(* CODESYS project mobject-graph-math-pack.library
   Company: mobject
   DefaultNamespace: mobject-graph-math-pack
   Version: 0.1.0
   Placeholder: mobject-graph-math-pack
   Author: mobject dev team
   Title: mobject-graph-math-pack

Project tree, tasks and I/O mapping:
  libraries: mobject-core, 0.7.0 (mobject); mobject-graph, 0.16.0 (mobject); Tc2_Math, * (Beckhoff Automation GmbH); Tc2_Standard, * (Beckhoff Automation GmbH); Tc2_System, * (Beckhoff Automation GmbH); Tc2_Utilities, * (Beckhoff Automation GmbH); Tc3_Module, * (Beckhoff Automation GmbH)
  Advanced/
    Nodes/
      ABS/
        function block ABS_BYTE [ST]: FB_init, Clone, OnExecute
        function block ABS_DINT [ST]: FB_init, Clone, OnExecute
        function block ABS_DWORD [ST]: FB_init, Clone, OnExecute
        function block ABS_INT [ST]: FB_init, Clone, OnExecute
        function block ABS_LINT [ST]: FB_init, Clone, OnExecute
        function block ABS_LREAL [ST]: FB_init, Clone, OnExecute
        function block ABS_LWORD [ST]: FB_init, Clone, OnExecute
        function block ABS_REAL [ST]: FB_init, Clone, OnExecute
        function block ABS_SINT [ST]: FB_init, Clone, OnExecute
        function block ABS_UDINT [ST]: FB_init, Clone, OnExecute
        function block ABS_UINT [ST]: FB_init, Clone, OnExecute
        function block ABS_ULINT [ST]: FB_init, Clone, OnExecute
        function block ABS_USINT [ST]: FB_init, Clone, OnExecute
        function block ABS_WORD [ST]: FB_init, Clone, OnExecute
      ACOS/
        function block ACOS_LREAL [ST]: FB_init, Clone, OnExecute
      ASIN/
        function block ASIN_LREAL [ST]: FB_init, Clone, OnExecute
      ATAN/
        function block ATAN_LREAL [ST]: FB_init, Clone, OnExecute
      COS/
        function block COS_LREAL [ST]: FB_init, Clone, OnExecute
      EXP/
        function block EXP_LREAL [ST]: FB_init, Clone, OnExecute
      EXPT/
        function block EXPT_LREAL [ST]: FB_init, Clone, OnExecute
      FLOOR/
        function block FLOOR_LREAL [ST]: FB_init, Clone, OnExecute
      FRAC/
        function block FRAC_LREAL [ST]: FB_init, Clone, OnExecute
      LN/
        function block LN_LREAL [ST]: FB_init, Clone, OnExecute
      LOG/
        function block LOG_LREAL [ST]: FB_init, Clone, OnExecute
      MODABS/
        function block MODABS_LREAL [ST]: FB_init, Clone, OnExecute
      MODTURNS/
        function block MODTURNS_LREAL [ST]: FB_init, Clone, OnExecute
      SIN/
        function block SIN_LREAL [ST]: FB_init, Clone, OnExecute
      SQRT/
        function block SQRT_LREAL [ST]: FB_init, Clone, OnExecute
      TAN/
        function block TAN_LREAL [ST]: FB_init, Clone, OnExecute
      TRUNC/
        function block TRUNC_LREAL [ST]: FB_init, Clone, OnExecute
      function block MathAdvancedPack [ST]: Register
  Comparison/
    Nodes/
      EQ/
        function block EQ_BYTE [ST]: FB_init, Clone, OnExecute
        function block EQ_DINT [ST]: FB_init, Clone, OnExecute
        function block EQ_DWORD [ST]: FB_init, Clone, OnExecute
        function block EQ_INT [ST]: FB_init, Clone, OnExecute
        function block EQ_LINT [ST]: FB_init, Clone, OnExecute
        function block EQ_LREAL [ST]: FB_init, Clone, OnExecute
        function block EQ_LWORD [ST]: FB_init, Clone, OnExecute
        function block EQ_REAL [ST]: FB_init, Clone, OnExecute
        function block EQ_SINT [ST]: FB_init, Clone, OnExecute
        function block EQ_UDINT [ST]: FB_init, Clone, OnExecute
        function block EQ_UINT [ST]: FB_init, Clone, OnExecute
        function block EQ_ULINT [ST]: FB_init, Clone, OnExecute
        function block EQ_USINT [ST]: FB_init, Clone, OnExecute
        function block EQ_WORD [ST]: FB_init, Clone, OnExecute
      GE/
        function block GE_BYTE [ST]: FB_init, Clone, OnExecute
        function block GE_DINT [ST]: FB_init, Clone, OnExecute
        function block GE_DWORD [ST]: FB_init, Clone, OnExecute
        function block GE_INT [ST]: FB_init, Clone, OnExecute
        function block GE_LINT [ST]: FB_init, Clone, OnExecute
        function block GE_LREAL [ST]: FB_init, Clone, OnExecute
        function block GE_LWORD [ST]: FB_init, Clone, OnExecute
        function block GE_REAL [ST]: FB_init, Clone, OnExecute
        function block GE_SINT [ST]: FB_init, Clone, OnExecute
        function block GE_UDINT [ST]: FB_init, Clone, OnExecute
        function block GE_UINT [ST]: FB_init, Clone, OnExecute
        function block GE_ULINT [ST]: FB_init, Clone, OnExecute
        function block GE_USINT [ST]: FB_init, Clone, OnExecute
        function block GE_WORD [ST]: FB_init, Clone, OnExecute
      GT/
        function block GT_BYTE [ST]: FB_init, Clone, OnExecute
        function block GT_DINT [ST]: FB_init, Clone, OnExecute
        function block GT_DWORD [ST]: FB_init, Clone, OnExecute
        function block GT_INT [ST]: FB_init, Clone, OnExecute
        function block GT_LINT [ST]: FB_init, Clone, OnExecute
        function block GT_LREAL [ST]: FB_init, Clone, OnExecute
        function block GT_LWORD [ST]: FB_init, Clone, OnExecute
        function block GT_REAL [ST]: FB_init, Clone, OnExecute
        function block GT_SINT [ST]: FB_init, Clone, OnExecute
        function block GT_UDINT [ST]: FB_init, Clone, OnExecute
        function block GT_UINT [ST]: FB_init, Clone, OnExecute
        function block GT_ULINT [ST]: FB_init, Clone, OnExecute
        function block GT_USINT [ST]: FB_init, Clone, OnExecute
        function block GT_WORD [ST]: FB_init, Clone, OnExecute
      LE/
        function block LE_BYTE [ST]: FB_init, Clone, OnExecute
        function block LE_DINT [ST]: FB_init, Clone, OnExecute
        function block LE_DWORD [ST]: FB_init, Clone, OnExecute
        function block LE_INT [ST]: FB_init, Clone, OnExecute
        function block LE_LINT [ST]: FB_init, Clone, OnExecute
        function block LE_LREAL [ST]: FB_init, Clone, OnExecute
        function block LE_LWORD [ST]: FB_init, Clone, OnExecute
        function block LE_REAL [ST]: FB_init, Clone, OnExecute
        function block LE_SINT [ST]: FB_init, Clone, OnExecute
        function block LE_UDINT [ST]: FB_init, Clone, OnExecute
        function block LE_UINT [ST]: FB_init, Clone, OnExecute
        function block LE_ULINT [ST]: FB_init, Clone, OnExecute
        function block LE_USINT [ST]: FB_init, Clone, OnExecute
        function block LE_WORD [ST]: FB_init, Clone, OnExecute
      LT/
        function block LT_BYTE [ST]: FB_init, Clone, OnExecute
        function block LT_DINT [ST]: FB_init, Clone, OnExecute
        function block LT_DWORD [ST]: FB_init, Clone, OnExecute
        function block LT_INT [ST]: FB_init, Clone, OnExecute
        function block LT_LINT [ST]: FB_init, Clone, OnExecute
        function block LT_LREAL [ST]: FB_init, Clone, OnExecute
        function block LT_LWORD [ST]: FB_init, Clone, OnExecute
        function block LT_REAL [ST]: FB_init, Clone, OnExecute
        function block LT_SINT [ST]: FB_init, Clone, OnExecute
        function block LT_UDINT [ST]: FB_init, Clone, OnExecute
        function block LT_UINT [ST]: FB_init, Clone, OnExecute
        function block LT_ULINT [ST]: FB_init, Clone, OnExecute
        function block LT_USINT [ST]: FB_init, Clone, OnExecute
        function block LT_WORD [ST]: FB_init, Clone, OnExecute
      NE/
        function block NE_BYTE [ST]: FB_init, Clone, OnExecute
        function block NE_DINT [ST]: FB_init, Clone, OnExecute
        function block NE_DWORD [ST]: FB_init, Clone, OnExecute
        function block NE_INT [ST]: FB_init, Clone, OnExecute
        function block NE_LINT [ST]: FB_init, Clone, OnExecute
        function block NE_LREAL [ST]: FB_init, Clone, OnExecute
        function block NE_LWORD [ST]: FB_init, Clone, OnExecute
        function block NE_REAL [ST]: FB_init, Clone, OnExecute
        function block NE_SINT [ST]: FB_init, Clone, OnExecute
        function block NE_UDINT [ST]: FB_init, Clone, OnExecute
        function block NE_UINT [ST]: FB_init, Clone, OnExecute
        function block NE_ULINT [ST]: FB_init, Clone, OnExecute
        function block NE_USINT [ST]: FB_init, Clone, OnExecute
        function block NE_WORD [ST]: FB_init, Clone, OnExecute
    function block MathComparisonPack [ST]: Register
  Core/
    Nodes/
      ADD/
        function block ADD_BYTE [ST]: FB_init, Clone, OnExecute
        function block ADD_DINT [ST]: FB_init, Clone, OnExecute
        function block ADD_DWORD [ST]: FB_init, Clone, OnExecute
        function block ADD_INT [ST]: FB_init, Clone, OnExecute
        function block ADD_LINT [ST]: FB_init, Clone, OnExecute
        function block ADD_LREAL [ST]: FB_init, Clone, OnExecute
        function block ADD_LWORD [ST]: FB_init, Clone, OnExecute
        function block ADD_REAL [ST]: FB_init, Clone, OnExecute
        function block ADD_SINT [ST]: FB_init, Clone, OnExecute
        function block ADD_UDINT [ST]: FB_init, Clone, OnExecute
        function block ADD_UINT [ST]: FB_init, Clone, OnExecute
        function block ADD_ULINT [ST]: FB_init, Clone, OnExecute
        function block ADD_USINT [ST]: FB_init, Clone, OnExecute
        function block ADD_WORD [ST]: FB_init, Clone, OnExecute
      DIV/
        function block DIV_BYTE [ST]: FB_init, Clone, OnExecute
        function block DIV_DINT [ST]: FB_init, Clone, OnExecute
        function block DIV_DWORD [ST]: FB_init, Clone, OnExecute
        function block DIV_INT [ST]: FB_init, Clone, OnExecute
        function block DIV_LINT [ST]: FB_init, Clone, OnExecute
        function block DIV_LREAL [ST]: FB_init, Clone, OnExecute
        function block DIV_LWORD [ST]: FB_init, Clone, OnExecute
        function block DIV_REAL [ST]: FB_init, Clone, OnExecute
        function block DIV_SINT [ST]: FB_init, Clone, OnExecute
        function block DIV_UDINT [ST]: FB_init, Clone, OnExecute
        function block DIV_UINT [ST]: FB_init, Clone, OnExecute
        function block DIV_ULINT [ST]: FB_init, Clone, OnExecute
        function block DIV_USINT [ST]: FB_init, Clone, OnExecute
        function block DIV_WORD [ST]: FB_init, Clone, OnExecute
      MOD/
        function block MOD_BYTE [ST]: FB_init, Clone, OnExecute
        function block MOD_DINT [ST]: FB_init, Clone, OnExecute
        function block MOD_DWORD [ST]: FB_init, Clone, OnExecute
        function block MOD_INT [ST]: FB_init, Clone, OnExecute
        function block MOD_LINT [ST]: FB_init, Clone, OnExecute
        function block MOD_LREAL [ST]: FB_init, Clone, OnExecute
        function block MOD_LWORD [ST]: FB_init, Clone, OnExecute
        function block MOD_SINT [ST]: FB_init, Clone, OnExecute
        function block MOD_UDINT [ST]: FB_init, Clone, OnExecute
        function block MOD_UINT [ST]: FB_init, Clone, OnExecute
        function block MOD_ULINT [ST]: FB_init, Clone, OnExecute
        function block MOD_USINT [ST]: FB_init, Clone, OnExecute
        function block MOD_WORD [ST]: FB_init, Clone, OnExecute
      MUL/
        function block MUL_BYTE [ST]: FB_init, Clone, OnExecute
        function block MUL_DINT [ST]: FB_init, Clone, OnExecute
        function block MUL_DWORD [ST]: FB_init, Clone, OnExecute
        function block MUL_INT [ST]: FB_init, Clone, OnExecute
        function block MUL_LINT [ST]: FB_init, Clone, OnExecute
        function block MUL_LREAL [ST]: FB_init, Clone, OnExecute
        function block MUL_LWORD [ST]: FB_init, Clone, OnExecute
        function block MUL_REAL [ST]: FB_init, Clone, OnExecute
        function block MUL_SINT [ST]: FB_init, Clone, OnExecute
        function block MUL_UDINT [ST]: FB_init, Clone, OnExecute
        function block MUL_UINT [ST]: FB_init, Clone, OnExecute
        function block MUL_ULINT [ST]: FB_init, Clone, OnExecute
        function block MUL_USINT [ST]: FB_init, Clone, OnExecute
        function block MUL_WORD [ST]: FB_init, Clone, OnExecute
      SUB/
        function block SUB_BYTE [ST]: FB_init, Clone, OnExecute
        function block SUB_DINT [ST]: FB_init, Clone, OnExecute
        function block SUB_DWORD [ST]: FB_init, Clone, OnExecute
        function block SUB_INT [ST]: FB_init, Clone, OnExecute
        function block SUB_LINT [ST]: FB_init, Clone, OnExecute
        function block SUB_LREAL [ST]: FB_init, Clone, OnExecute
        function block SUB_LWORD [ST]: FB_init, Clone, OnExecute
        function block SUB_REAL [ST]: FB_init, Clone, OnExecute
        function block SUB_SINT [ST]: FB_init, Clone, OnExecute
        function block SUB_UDINT [ST]: FB_init, Clone, OnExecute
        function block SUB_UINT [ST]: FB_init, Clone, OnExecute
        function block SUB_ULINT [ST]: FB_init, Clone, OnExecute
        function block SUB_USINT [ST]: FB_init, Clone, OnExecute
        function block SUB_WORD [ST]: FB_init, Clone, OnExecute
    function block MathCorePack [ST]: Register
  Logic/
    Nodes/
      AND/
        function block AND_BOOL [ST]: FB_init, Clone, OnExecute
        function block AND_BYTE [ST]: FB_init, Clone, OnExecute
        function block AND_DINT [ST]: FB_init, Clone, OnExecute
        function block AND_DWORD [ST]: FB_init, Clone, OnExecute
        function block AND_INT [ST]: FB_init, Clone, OnExecute
        function block AND_LINT [ST]: FB_init, Clone, OnExecute
        function block AND_LWORD [ST]: FB_init, Clone, OnExecute
        function block AND_SINT [ST]: FB_init, Clone, OnExecute
        function block AND_UDINT [ST]: FB_init, Clone, OnExecute
        function block AND_UINT [ST]: FB_init, Clone, OnExecute
        function block AND_ULINT [ST]: FB_init, Clone, OnExecute
        function block AND_USINT [ST]: FB_init, Clone, OnExecute
        function block AND_WORD [ST]: FB_init, Clone, OnExecute
      NOT/
        function block NOT_BOOL [ST]: FB_init, Clone, OnExecute
        function block NOT_BYTE [ST]: FB_init, Clone, OnExecute
        function block NOT_DINT [ST]: FB_init, Clone, OnExecute
        function block NOT_DWORD [ST]: FB_init, Clone, OnExecute
        function block NOT_INT [ST]: FB_init, Clone, OnExecute
        function block NOT_LINT [ST]: FB_init, Clone, OnExecute
        function block NOT_LWORD [ST]: FB_init, Clone, OnExecute
        function block NOT_SINT [ST]: FB_init, Clone, OnExecute
        function block NOT_UDINT [ST]: FB_init, Clone, OnExecute
        function block NOT_UINT [ST]: FB_init, Clone, OnExecute
        function block NOT_ULINT [ST]: FB_init, Clone, OnExecute
        function block NOT_USINT [ST]: FB_init, Clone, OnExecute
        function block NOT_WORD [ST]: FB_init, Clone, OnExecute
      OR/
        function block OR_BOOL [ST]: FB_init, Clone, OnExecute
        function block OR_BYTE [ST]: FB_init, Clone, OnExecute
        function block OR_DINT [ST]: FB_init, Clone, OnExecute
        function block OR_DWORD [ST]: FB_init, Clone, OnExecute
        function block OR_INT [ST]: FB_init, Clone, OnExecute
        function block OR_LINT [ST]: FB_init, Clone, OnExecute
        function block OR_LWORD [ST]: FB_init, Clone, OnExecute
        function block OR_SINT [ST]: FB_init, Clone, OnExecute
        function block OR_UDINT [ST]: FB_init, Clone, OnExecute
        function block OR_UINT [ST]: FB_init, Clone, OnExecute
        function block OR_ULINT [ST]: FB_init, Clone, OnExecute
        function block OR_USINT [ST]: FB_init, Clone, OnExecute
        function block OR_WORD [ST]: FB_init, Clone, OnExecute
      XOR/
        function block XOR_BOOL [ST]: FB_init, Clone, OnExecute
        function block XOR_BYTE [ST]: FB_init, Clone, OnExecute
        function block XOR_DINT [ST]: FB_init, Clone, OnExecute
        function block XOR_DWORD [ST]: FB_init, Clone, OnExecute
        function block XOR_INT [ST]: FB_init, Clone, OnExecute
        function block XOR_LINT [ST]: FB_init, Clone, OnExecute
        function block XOR_LWORD [ST]: FB_init, Clone, OnExecute
        function block XOR_SINT [ST]: FB_init, Clone, OnExecute
        function block XOR_UDINT [ST]: FB_init, Clone, OnExecute
        function block XOR_UINT [ST]: FB_init, Clone, OnExecute
        function block XOR_ULINT [ST]: FB_init, Clone, OnExecute
        function block XOR_USINT [ST]: FB_init, Clone, OnExecute
        function block XOR_WORD [ST]: FB_init, Clone, OnExecute
    function block MathLogicPack [ST]: Register
  Selection/
    Nodes/
      MAX/
        function block MAX_BYTE [ST]: FB_init, Clone, OnExecute
        function block MAX_DINT [ST]: FB_init, Clone, OnExecute
        function block MAX_DWORD [ST]: FB_init, Clone, OnExecute
        function block MAX_INT [ST]: FB_init, Clone, OnExecute
        function block MAX_LINT [ST]: FB_init, Clone, OnExecute
        function block MAX_LREAL [ST]: FB_init, Clone, OnExecute
        function block MAX_LWORD [ST]: FB_init, Clone, OnExecute
        function block MAX_REAL [ST]: FB_init, Clone, OnExecute
        function block MAX_SINT [ST]: FB_init, Clone, OnExecute
        function block MAX_UDINT [ST]: FB_init, Clone, OnExecute
        function block MAX_UINT [ST]: FB_init, Clone, OnExecute
        function block MAX_ULINT [ST]: FB_init, Clone, OnExecute
        function block MAX_USINT [ST]: FB_init, Clone, OnExecute
        function block MAX_WORD [ST]: FB_init, Clone, OnExecute
      MIN/
        function block MIN_BYTE [ST]: FB_init, Clone, OnExecute
        function block MIN_DINT [ST]: FB_init, Clone, OnExecute
        function block MIN_DWORD [ST]: FB_init, Clone, OnExecute
        function block MIN_INT [ST]: FB_init, Clone, OnExecute
        function block MIN_LINT [ST]: FB_init, Clone, OnExecute
        function block MIN_LREAL [ST]: FB_init, Clone, OnExecute
        function block MIN_LWORD [ST]: FB_init, Clone, OnExecute
        function block MIN_REAL [ST]: FB_init, Clone, OnExecute
        function block MIN_SINT [ST]: FB_init, Clone, OnExecute
        function block MIN_UDINT [ST]: FB_init, Clone, OnExecute
        function block MIN_UINT [ST]: FB_init, Clone, OnExecute
        function block MIN_ULINT [ST]: FB_init, Clone, OnExecute
        function block MIN_USINT [ST]: FB_init, Clone, OnExecute
        function block MIN_WORD [ST]: FB_init, Clone, OnExecute
      SEL/
        function block SEL_BYTE [ST]: FB_init, Clone, OnExecute
        function block SEL_DINT [ST]: FB_init, Clone, OnExecute
        function block SEL_DWORD [ST]: FB_init, Clone, OnExecute
        function block SEL_INT [ST]: FB_init, Clone, OnExecute
        function block SEL_LINT [ST]: FB_init, Clone, OnExecute
        function block SEL_LREAL [ST]: FB_init, Clone, OnExecute
        function block SEL_LWORD [ST]: FB_init, Clone, OnExecute
        function block SEL_REAL [ST]: FB_init, Clone, OnExecute
        function block SEL_SINT [ST]: FB_init, Clone, OnExecute
        function block SEL_UDINT [ST]: FB_init, Clone, OnExecute
        function block SEL_UINT [ST]: FB_init, Clone, OnExecute
        function block SEL_ULINT [ST]: FB_init, Clone, OnExecute
        function block SEL_USINT [ST]: FB_init, Clone, OnExecute
        function block SEL_WORD [ST]: FB_init, Clone, OnExecute
    function block MathSelectionPack [ST]: Register
  function block MathPack [ST]: Register
*)

// Advanced/Nodes/ABS/ABS_BYTE
{attribute 'linkalways'} 
{attribute 'no_explicit_call' := 'This FB is a CLASS and must be accessed using methods or properties'}
{attribute 'enable_dynamic_creation'}
FUNCTION_BLOCK FINAL ABS_BYTE EXTENDS Node
VAR
	in : _BYTE(0);
	out : _BYTE(0);
END_VAR

METHOD FB_init : BOOL
VAR_INPUT
	bInitRetains : BOOL; // if TRUE, the retain variables are initialized (warm start / cold start)
	bInCopyCode : BOOL;  // if TRUE, the instance afterwards gets moved into the copy code (online change)
END_VAR
AddInput('in',THIS^.in);
AddOutput('out', THIS^.out);
END_METHOD

METHOD PUBLIC Clone : I_Node
VAR
	pNode : POINTER TO ABS_BYTE;
END_VAR
pNode := __NEW(ABS_BYTE);
Clone := pNode^;
END_METHOD

METHOD PROTECTED OnExecute
VAR
END_VAR
out.Value := ABS(in.Value);
END_METHOD

END_FUNCTION_BLOCK

// Advanced/Nodes/ABS/ABS_DINT
{attribute 'linkalways'} 
{attribute 'no_explicit_call' := 'This FB is a CLASS and must be accessed using methods or properties'}
{attribute 'enable_dynamic_creation'}
FUNCTION_BLOCK FINAL ABS_DINT EXTENDS Node
VAR
	in : _DINT(0);
	out : _DINT(0);
END_VAR

METHOD FB_init : BOOL
VAR_INPUT
	bInitRetains : BOOL; // if TRUE, the retain variables are initialized (warm start / cold start)
	bInCopyCode : BOOL;  // if TRUE, the instance afterwards gets moved into the copy code (online change)
END_VAR
AddInput('in',THIS^.in);
AddOutput('out', THIS^.out);
END_METHOD

METHOD PUBLIC Clone : I_Node
VAR
	pNode : POINTER TO ABS_DINT;
END_VAR
pNode := __NEW(ABS_DINT);
Clone := pNode^;
END_METHOD

METHOD PROTECTED OnExecute
VAR
END_VAR
out.Value := ABS(in.Value);
END_METHOD

END_FUNCTION_BLOCK

// Advanced/Nodes/ABS/ABS_DWORD
{attribute 'linkalways'} 
{attribute 'no_explicit_call' := 'This FB is a CLASS and must be accessed using methods or properties'}
{attribute 'enable_dynamic_creation'}
FUNCTION_BLOCK FINAL ABS_DWORD EXTENDS Node
VAR
	in : _DWORD(0);
	out : _DWORD(0);
END_VAR

METHOD FB_init : BOOL
VAR_INPUT
	bInitRetains : BOOL; // if TRUE, the retain variables are initialized (warm start / cold start)
	bInCopyCode : BOOL;  // if TRUE, the instance afterwards gets moved into the copy code (online change)
END_VAR
AddInput('in',THIS^.in);
AddOutput('out', THIS^.out);
END_METHOD

METHOD PUBLIC Clone : I_Node
VAR
	pNode : POINTER TO ABS_DWORD;
END_VAR
pNode := __NEW(ABS_DWORD);
Clone := pNode^;
END_METHOD

METHOD PROTECTED OnExecute
VAR
END_VAR
out.Value := ABS(in.Value);
END_METHOD

END_FUNCTION_BLOCK

// Advanced/Nodes/ABS/ABS_INT
{attribute 'linkalways'} 
{attribute 'no_explicit_call' := 'This FB is a CLASS and must be accessed using methods or properties'}
{attribute 'enable_dynamic_creation'}
FUNCTION_BLOCK FINAL ABS_INT EXTENDS Node
VAR
	in : _INT(0);
	out : _INT(0);
END_VAR

METHOD FB_init : BOOL
VAR_INPUT
	bInitRetains : BOOL; // if TRUE, the retain variables are initialized (warm start / cold start)
	bInCopyCode : BOOL;  // if TRUE, the instance afterwards gets moved into the copy code (online change)
END_VAR
AddInput('in',THIS^.in);
AddOutput('out', THIS^.out);
END_METHOD

METHOD PUBLIC Clone : I_Node
VAR
	pNode : POINTER TO ABS_INT;
END_VAR
pNode := __NEW(ABS_INT);
Clone := pNode^;
END_METHOD

METHOD PROTECTED OnExecute
VAR
END_VAR
out.Value := ABS(in.Value);
END_METHOD

END_FUNCTION_BLOCK

// Advanced/Nodes/ABS/ABS_LINT
{attribute 'linkalways'} 
{attribute 'no_explicit_call' := 'This FB is a CLASS and must be accessed using methods or properties'}
{attribute 'enable_dynamic_creation'}
FUNCTION_BLOCK FINAL ABS_LINT EXTENDS Node
VAR
	in : _LINT(0);
	out : _LINT(0);
END_VAR

METHOD FB_init : BOOL
VAR_INPUT
	bInitRetains : BOOL; // if TRUE, the retain variables are initialized (warm start / cold start)
	bInCopyCode : BOOL;  // if TRUE, the instance afterwards gets moved into the copy code (online change)
END_VAR
AddInput('in',THIS^.in);
AddOutput('out', THIS^.out);
END_METHOD

METHOD PUBLIC Clone : I_Node
VAR
	pNode : POINTER TO ABS_LINT;
END_VAR
pNode := __NEW(ABS_LINT);
Clone := pNode^;
END_METHOD

METHOD PROTECTED OnExecute
VAR
END_VAR
out.Value := ABS(in.Value);
END_METHOD

END_FUNCTION_BLOCK

// Advanced/Nodes/ABS/ABS_LREAL
{attribute 'linkalways'} 
{attribute 'no_explicit_call' := 'This FB is a CLASS and must be accessed using methods or properties'}
{attribute 'enable_dynamic_creation'}
FUNCTION_BLOCK FINAL ABS_LREAL EXTENDS Node
VAR
	in : _LREAL(0.0);
	out : _LREAL(0.0);
END_VAR

METHOD FB_init : BOOL
VAR_INPUT
	bInitRetains : BOOL; // if TRUE, the retain variables are initialized (warm start / cold start)
	bInCopyCode : BOOL;  // if TRUE, the instance afterwards gets moved into the copy code (online change)
END_VAR
AddInput('in',THIS^.in);
AddOutput('out', THIS^.out);
END_METHOD

METHOD PUBLIC Clone : I_Node
VAR
	pNode : POINTER TO ABS_LREAL;
END_VAR
pNode := __NEW(ABS_LREAL);
Clone := pNode^;
END_METHOD

METHOD PROTECTED OnExecute
VAR
END_VAR
out.Value := ABS(in.Value);
END_METHOD

END_FUNCTION_BLOCK

// Advanced/Nodes/ABS/ABS_LWORD
{attribute 'linkalways'} 
{attribute 'no_explicit_call' := 'This FB is a CLASS and must be accessed using methods or properties'}
{attribute 'enable_dynamic_creation'}
FUNCTION_BLOCK FINAL ABS_LWORD EXTENDS Node
VAR
	in : _LWORD(0);
	out : _LWORD(0);
END_VAR

METHOD FB_init : BOOL
VAR_INPUT
	bInitRetains : BOOL; // if TRUE, the retain variables are initialized (warm start / cold start)
	bInCopyCode : BOOL;  // if TRUE, the instance afterwards gets moved into the copy code (online change)
END_VAR
AddInput('in',THIS^.in);
AddOutput('out', THIS^.out);
END_METHOD

METHOD PUBLIC Clone : I_Node
VAR
	pNode : POINTER TO ABS_LWORD;
END_VAR
pNode := __NEW(ABS_LWORD);
Clone := pNode^;
END_METHOD

METHOD PROTECTED OnExecute
VAR
END_VAR
out.Value := ABS(in.Value);
END_METHOD

END_FUNCTION_BLOCK

// Advanced/Nodes/ABS/ABS_REAL
{attribute 'linkalways'} 
{attribute 'no_explicit_call' := 'This FB is a CLASS and must be accessed using methods or properties'}
{attribute 'enable_dynamic_creation'}
FUNCTION_BLOCK FINAL ABS_REAL EXTENDS Node
VAR
	in : _REAL(0.0);
	out : _REAL(0.0);
END_VAR

METHOD FB_init : BOOL
VAR_INPUT
	bInitRetains : BOOL; // if TRUE, the retain variables are initialized (warm start / cold start)
	bInCopyCode : BOOL;  // if TRUE, the instance afterwards gets moved into the copy code (online change)
END_VAR
AddInput('in',THIS^.in);
AddOutput('out', THIS^.out);
END_METHOD

METHOD PUBLIC Clone : I_Node
VAR
	pNode : POINTER TO ABS_REAL;
END_VAR
pNode := __NEW(ABS_REAL);
Clone := pNode^;
END_METHOD

METHOD PROTECTED OnExecute
VAR
END_VAR
out.Value := ABS(in.Value);
END_METHOD

END_FUNCTION_BLOCK

// Advanced/Nodes/ABS/ABS_SINT
{attribute 'linkalways'} 
{attribute 'no_explicit_call' := 'This FB is a CLASS and must be accessed using methods or properties'}
{attribute 'enable_dynamic_creation'}
FUNCTION_BLOCK FINAL ABS_SINT EXTENDS Node
VAR
	in : _SINT(0);
	out : _SINT(0);
END_VAR

METHOD FB_init : BOOL
VAR_INPUT
	bInitRetains : BOOL; // if TRUE, the retain variables are initialized (warm start / cold start)
	bInCopyCode : BOOL;  // if TRUE, the instance afterwards gets moved into the copy code (online change)
END_VAR
AddInput('in',THIS^.in);
AddOutput('out', THIS^.out);
END_METHOD

METHOD PUBLIC Clone : I_Node
VAR
	pNode : POINTER TO ABS_SINT;
END_VAR
pNode := __NEW(ABS_SINT);
Clone := pNode^;
END_METHOD

METHOD PROTECTED OnExecute
VAR
END_VAR
out.Value := ABS(in.Value);
END_METHOD

END_FUNCTION_BLOCK

// Advanced/Nodes/ABS/ABS_UDINT
{attribute 'linkalways'} 
{attribute 'no_explicit_call' := 'This FB is a CLASS and must be accessed using methods or properties'}
{attribute 'enable_dynamic_creation'}
FUNCTION_BLOCK FINAL ABS_UDINT EXTENDS Node
VAR
	in : _UDINT(0);
	out : _UDINT(0);
END_VAR

METHOD FB_init : BOOL
VAR_INPUT
	bInitRetains : BOOL; // if TRUE, the retain variables are initialized (warm start / cold start)
	bInCopyCode : BOOL;  // if TRUE, the instance afterwards gets moved into the copy code (online change)
END_VAR
AddInput('in',THIS^.in);
AddOutput('out', THIS^.out);
END_METHOD

METHOD PUBLIC Clone : I_Node
VAR
	pNode : POINTER TO ABS_UDINT;
END_VAR
pNode := __NEW(ABS_UDINT);
Clone := pNode^;
END_METHOD

METHOD PROTECTED OnExecute
VAR
END_VAR
out.Value := ABS(in.Value);
END_METHOD

END_FUNCTION_BLOCK

// Advanced/Nodes/ABS/ABS_UINT
{attribute 'linkalways'} 
{attribute 'no_explicit_call' := 'This FB is a CLASS and must be accessed using methods or properties'}
{attribute 'enable_dynamic_creation'}
FUNCTION_BLOCK FINAL ABS_UINT EXTENDS Node
VAR
	in : _UINT(0);
	out : _UINT(0);
END_VAR

METHOD FB_init : BOOL
VAR_INPUT
	bInitRetains : BOOL; // if TRUE, the retain variables are initialized (warm start / cold start)
	bInCopyCode : BOOL;  // if TRUE, the instance afterwards gets moved into the copy code (online change)
END_VAR
AddInput('in',THIS^.in);
AddOutput('out', THIS^.out);
END_METHOD

METHOD PUBLIC Clone : I_Node
VAR
	pNode : POINTER TO ABS_UINT;
END_VAR
pNode := __NEW(ABS_UINT);
Clone := pNode^;
END_METHOD

METHOD PROTECTED OnExecute
VAR
END_VAR
out.Value := ABS(in.Value);
END_METHOD

END_FUNCTION_BLOCK

// Advanced/Nodes/ABS/ABS_ULINT
{attribute 'linkalways'} 
{attribute 'no_explicit_call' := 'This FB is a CLASS and must be accessed using methods or properties'}
{attribute 'enable_dynamic_creation'}
FUNCTION_BLOCK FINAL ABS_ULINT EXTENDS Node
VAR
	in : _ULINT(0);
	out : _ULINT(0);
END_VAR

METHOD FB_init : BOOL
VAR_INPUT
	bInitRetains : BOOL; // if TRUE, the retain variables are initialized (warm start / cold start)
	bInCopyCode : BOOL;  // if TRUE, the instance afterwards gets moved into the copy code (online change)
END_VAR
AddInput('in',THIS^.in);
AddOutput('out', THIS^.out);
END_METHOD

METHOD PUBLIC Clone : I_Node
VAR
	pNode : POINTER TO ABS_ULINT;
END_VAR
pNode := __NEW(ABS_ULINT);
Clone := pNode^;
END_METHOD

METHOD PROTECTED OnExecute
VAR
END_VAR
out.Value := ABS(in.Value);
END_METHOD

END_FUNCTION_BLOCK

// Advanced/Nodes/ABS/ABS_USINT
{attribute 'linkalways'} 
{attribute 'no_explicit_call' := 'This FB is a CLASS and must be accessed using methods or properties'}
{attribute 'enable_dynamic_creation'}
FUNCTION_BLOCK FINAL ABS_USINT EXTENDS Node
VAR
	in : _USINT(0);
	out : _USINT(0);
END_VAR

METHOD FB_init : BOOL
VAR_INPUT
	bInitRetains : BOOL; // if TRUE, the retain variables are initialized (warm start / cold start)
	bInCopyCode : BOOL;  // if TRUE, the instance afterwards gets moved into the copy code (online change)
END_VAR
AddInput('in',THIS^.in);
AddOutput('out', THIS^.out);
END_METHOD

METHOD PUBLIC Clone : I_Node
VAR
	pNode : POINTER TO ABS_USINT;
END_VAR
pNode := __NEW(ABS_USINT);
Clone := pNode^;
END_METHOD

METHOD PROTECTED OnExecute
VAR
END_VAR
out.Value := ABS(in.Value);
END_METHOD

END_FUNCTION_BLOCK

// Advanced/Nodes/ABS/ABS_WORD
{attribute 'linkalways'} 
{attribute 'no_explicit_call' := 'This FB is a CLASS and must be accessed using methods or properties'}
{attribute 'enable_dynamic_creation'}
FUNCTION_BLOCK FINAL ABS_WORD EXTENDS Node
VAR
	in : _WORD(0);
	out : _WORD(0);
END_VAR

METHOD FB_init : BOOL
VAR_INPUT
	bInitRetains : BOOL; // if TRUE, the retain variables are initialized (warm start / cold start)
	bInCopyCode : BOOL;  // if TRUE, the instance afterwards gets moved into the copy code (online change)
END_VAR
AddInput('in',THIS^.in);
AddOutput('out', THIS^.out);
END_METHOD

METHOD PUBLIC Clone : I_Node
VAR
	pNode : POINTER TO ABS_WORD;
END_VAR
pNode := __NEW(ABS_WORD);
Clone := pNode^;
END_METHOD

METHOD PROTECTED OnExecute
VAR
END_VAR
out.Value := ABS(in.Value);
END_METHOD

END_FUNCTION_BLOCK

// Advanced/Nodes/ACOS/ACOS_LREAL
{attribute 'linkalways'} 
{attribute 'no_explicit_call' := 'This FB is a CLASS and must be accessed using methods or properties'}
{attribute 'enable_dynamic_creation'}
FUNCTION_BLOCK FINAL ACOS_LREAL EXTENDS Node
VAR
	in : _LREAL(0.0);
	out : _LREAL(0.0);
END_VAR

METHOD FB_init : BOOL
VAR_INPUT
	bInitRetains : BOOL; // if TRUE, the retain variables are initialized (warm start / cold start)
	bInCopyCode : BOOL;  // if TRUE, the instance afterwards gets moved into the copy code (online change)
END_VAR
AddInput('in',THIS^.in);
AddOutput('out', THIS^.out);
END_METHOD

METHOD PUBLIC Clone : I_Node
VAR
	pNode : POINTER TO ACOS_LREAL;
END_VAR
pNode := __NEW(ACOS_LREAL);
Clone := pNode^;
END_METHOD

METHOD PROTECTED OnExecute
VAR
END_VAR
out.Value := ACOS(in.Value);
END_METHOD

END_FUNCTION_BLOCK

// Advanced/Nodes/ASIN/ASIN_LREAL
{attribute 'linkalways'} 
{attribute 'no_explicit_call' := 'This FB is a CLASS and must be accessed using methods or properties'}
{attribute 'enable_dynamic_creation'}
FUNCTION_BLOCK FINAL ASIN_LREAL EXTENDS Node
VAR
	in : _LREAL(0.0);
	out : _LREAL(0.0);
END_VAR

METHOD FB_init : BOOL
VAR_INPUT
	bInitRetains : BOOL; // if TRUE, the retain variables are initialized (warm start / cold start)
	bInCopyCode : BOOL;  // if TRUE, the instance afterwards gets moved into the copy code (online change)
END_VAR
AddInput('in',THIS^.in);
AddOutput('out', THIS^.out);
END_METHOD

METHOD PUBLIC Clone : I_Node
VAR
	pNode : POINTER TO ASIN_LREAL;
END_VAR
pNode := __NEW(ASIN_LREAL);
Clone := pNode^;
END_METHOD

METHOD PROTECTED OnExecute
VAR
END_VAR
out.Value := ASIN(in.Value);
END_METHOD

END_FUNCTION_BLOCK

// Advanced/Nodes/ATAN/ATAN_LREAL
{attribute 'linkalways'} 
{attribute 'no_explicit_call' := 'This FB is a CLASS and must be accessed using methods or properties'}
{attribute 'enable_dynamic_creation'}
FUNCTION_BLOCK FINAL ATAN_LREAL EXTENDS Node
VAR
	in : _LREAL(0.0);
	out : _LREAL(0.0);
END_VAR

METHOD FB_init : BOOL
VAR_INPUT
	bInitRetains : BOOL; // if TRUE, the retain variables are initialized (warm start / cold start)
	bInCopyCode : BOOL;  // if TRUE, the instance afterwards gets moved into the copy code (online change)
END_VAR
AddInput('in',THIS^.in);
AddOutput('out', THIS^.out);
END_METHOD

METHOD PUBLIC Clone : I_Node
VAR
	pNode : POINTER TO ATAN_LREAL;
END_VAR
pNode := __NEW(ATAN_LREAL);
Clone := pNode^;
END_METHOD

METHOD PROTECTED OnExecute
VAR
END_VAR
out.Value := ATAN(in.Value);
END_METHOD

END_FUNCTION_BLOCK

// Advanced/Nodes/COS/COS_LREAL
{attribute 'linkalways'} 
{attribute 'no_explicit_call' := 'This FB is a CLASS and must be accessed using methods or properties'}
{attribute 'enable_dynamic_creation'}
FUNCTION_BLOCK FINAL COS_LREAL EXTENDS Node
VAR
	in : _LREAL(0.0);
	out : _LREAL(0.0);
END_VAR

METHOD FB_init : BOOL
VAR_INPUT
	bInitRetains : BOOL; // if TRUE, the retain variables are initialized (warm start / cold start)
	bInCopyCode : BOOL;  // if TRUE, the instance afterwards gets moved into the copy code (online change)
END_VAR
AddInput('in',THIS^.in);
AddOutput('out', THIS^.out);
END_METHOD

METHOD PUBLIC Clone : I_Node
VAR
	pNode : POINTER TO COS_LREAL;
END_VAR
pNode := __NEW(COS_LREAL);
Clone := pNode^;
END_METHOD

METHOD PROTECTED OnExecute
VAR
END_VAR
out.Value := COS(in.Value);
END_METHOD

END_FUNCTION_BLOCK

// Advanced/Nodes/EXP/EXP_LREAL
{attribute 'linkalways'} 
{attribute 'no_explicit_call' := 'This FB is a CLASS and must be accessed using methods or properties'}
{attribute 'enable_dynamic_creation'}
FUNCTION_BLOCK FINAL EXP_LREAL EXTENDS Node
VAR
	in : _LREAL(0.0);
	out : _LREAL(0.0);
END_VAR

METHOD FB_init : BOOL
VAR_INPUT
	bInitRetains : BOOL; // if TRUE, the retain variables are initialized (warm start / cold start)
	bInCopyCode : BOOL;  // if TRUE, the instance afterwards gets moved into the copy code (online change)
END_VAR
AddInput('in',THIS^.in);
AddOutput('out', THIS^.out);
END_METHOD

METHOD PUBLIC Clone : I_Node
VAR
	pNode : POINTER TO EXP_LREAL;
END_VAR
pNode := __NEW(EXP_LREAL);
Clone := pNode^;
END_METHOD

METHOD PROTECTED OnExecute
VAR
END_VAR
out.Value := EXP(in.Value);
END_METHOD

END_FUNCTION_BLOCK

// Advanced/Nodes/EXPT/EXPT_LREAL
{attribute 'linkalways'} 
{attribute 'no_explicit_call' := 'This FB is a CLASS and must be accessed using methods or properties'}
{attribute 'enable_dynamic_creation'}
FUNCTION_BLOCK FINAL EXPT_LREAL EXTENDS Node
VAR
	base : _LREAL(0.0);
	exponent : _LREAL(0.0);
	out : _LREAL(0.0);
END_VAR

METHOD FB_init : BOOL
VAR_INPUT
	bInitRetains : BOOL; // if TRUE, the retain variables are initialized (warm start / cold start)
	bInCopyCode : BOOL;  // if TRUE, the instance afterwards gets moved into the copy code (online change)
END_VAR
AddInput('base',THIS^.base);
AddInput('exponent',THIS^.exponent);
AddOutput('out', THIS^.out);
END_METHOD

METHOD PUBLIC Clone : I_Node
VAR
	pNode : POINTER TO EXPT_LREAL;
END_VAR
pNode := __NEW(EXPT_LREAL);
Clone := pNode^;
END_METHOD

METHOD PROTECTED OnExecute
VAR
END_VAR
out.Value := EXPT(base.Value, exponent.Value);
END_METHOD

END_FUNCTION_BLOCK

// Advanced/Nodes/FLOOR/FLOOR_LREAL
{attribute 'linkalways'} 
{attribute 'no_explicit_call' := 'This FB is a CLASS and must be accessed using methods or properties'}
{attribute 'enable_dynamic_creation'}
FUNCTION_BLOCK FINAL FLOOR_LREAL EXTENDS Node
VAR
	in : _LREAL(0.0);
	out : _LREAL(0.0);
END_VAR

METHOD FB_init : BOOL
VAR_INPUT
	bInitRetains : BOOL; // if TRUE, the retain variables are initialized (warm start / cold start)
	bInCopyCode : BOOL;  // if TRUE, the instance afterwards gets moved into the copy code (online change)
END_VAR
AddInput('in',THIS^.in);
AddOutput('out', THIS^.out);
END_METHOD

METHOD PUBLIC Clone : I_Node
VAR
	pNode : POINTER TO FLOOR_LREAL;
END_VAR
pNode := __NEW(FLOOR_LREAL);
Clone := pNode^;
END_METHOD

METHOD PROTECTED OnExecute
VAR
END_VAR
out.Value := FLOOR(in.Value);
END_METHOD

END_FUNCTION_BLOCK

// Advanced/Nodes/FRAC/FRAC_LREAL
{attribute 'linkalways'} 
{attribute 'no_explicit_call' := 'This FB is a CLASS and must be accessed using methods or properties'}
{attribute 'enable_dynamic_creation'}
FUNCTION_BLOCK FINAL FRAC_LREAL EXTENDS Node
VAR
	in : _LREAL(0.0);
	out : _LREAL(0.0);
END_VAR

METHOD FB_init : BOOL
VAR_INPUT
	bInitRetains : BOOL; // if TRUE, the retain variables are initialized (warm start / cold start)
	bInCopyCode : BOOL;  // if TRUE, the instance afterwards gets moved into the copy code (online change)
END_VAR
AddInput('in',THIS^.in);
AddOutput('out', THIS^.out);
END_METHOD

METHOD PUBLIC Clone : I_Node
VAR
	pNode : POINTER TO FRAC_LREAL;
END_VAR
pNode := __NEW(FRAC_LREAL);
Clone := pNode^;
END_METHOD

METHOD PROTECTED OnExecute
VAR
END_VAR
out.Value := FRAC(in.Value);
END_METHOD

END_FUNCTION_BLOCK

// Advanced/Nodes/LN/LN_LREAL
{attribute 'linkalways'} 
{attribute 'no_explicit_call' := 'This FB is a CLASS and must be accessed using methods or properties'}
{attribute 'enable_dynamic_creation'}
FUNCTION_BLOCK FINAL LN_LREAL EXTENDS Node
VAR
	in : _LREAL(0.0);
	out : _LREAL(0.0);
END_VAR

METHOD FB_init : BOOL
VAR_INPUT
	bInitRetains : BOOL; // if TRUE, the retain variables are initialized (warm start / cold start)
	bInCopyCode : BOOL;  // if TRUE, the instance afterwards gets moved into the copy code (online change)
END_VAR
AddInput('in',THIS^.in);
AddOutput('out', THIS^.out);
END_METHOD

METHOD PUBLIC Clone : I_Node
VAR
	pNode : POINTER TO LN_LREAL;
END_VAR
pNode := __NEW(LN_LREAL);
Clone := pNode^;
END_METHOD

METHOD PROTECTED OnExecute
VAR
END_VAR
out.Value := LN(in.Value);
END_METHOD

END_FUNCTION_BLOCK

// Advanced/Nodes/LOG/LOG_LREAL
{attribute 'linkalways'} 
{attribute 'no_explicit_call' := 'This FB is a CLASS and must be accessed using methods or properties'}
{attribute 'enable_dynamic_creation'}
FUNCTION_BLOCK FINAL LOG_LREAL EXTENDS Node
VAR
	in : _LREAL(0.0);
	out : _LREAL(0.0);
END_VAR

METHOD FB_init : BOOL
VAR_INPUT
	bInitRetains : BOOL; // if TRUE, the retain variables are initialized (warm start / cold start)
	bInCopyCode : BOOL;  // if TRUE, the instance afterwards gets moved into the copy code (online change)
END_VAR
AddInput('in',THIS^.in);
AddOutput('out', THIS^.out);
END_METHOD

METHOD PUBLIC Clone : I_Node
VAR
	pNode : POINTER TO LOG_LREAL;
END_VAR
pNode := __NEW(LOG_LREAL);
Clone := pNode^;
END_METHOD

METHOD PROTECTED OnExecute
VAR
END_VAR
out.Value := LOG(in.Value);
END_METHOD

END_FUNCTION_BLOCK

// Advanced/Nodes/MODABS/MODABS_LREAL
{attribute 'linkalways'} 
{attribute 'no_explicit_call' := 'This FB is a CLASS and must be accessed using methods or properties'}
{attribute 'enable_dynamic_creation'}
FUNCTION_BLOCK FINAL MODABS_LREAL EXTENDS Node
VAR
	value : _LREAL(0.0);
	arg : _LREAL(0.0);
	out : _LREAL(0.0);
END_VAR

METHOD FB_init : BOOL
VAR_INPUT
	bInitRetains : BOOL; // if TRUE, the retain variables are initialized (warm start / cold start)
	bInCopyCode : BOOL;  // if TRUE, the instance afterwards gets moved into the copy code (online change)
END_VAR
AddInput('value',THIS^.value);
AddInput('arg',THIS^.arg);
AddOutput('out', THIS^.out);
END_METHOD

METHOD PUBLIC Clone : I_Node
VAR
	pNode : POINTER TO MODABS_LREAL;
END_VAR
pNode := __NEW(MODABS_LREAL);
Clone := pNode^;
END_METHOD

METHOD PROTECTED OnExecute
VAR
END_VAR
out.Value := MODABS(value.Value, arg.Value);
END_METHOD

END_FUNCTION_BLOCK

// Advanced/Nodes/MODTURNS/MODTURNS_LREAL
{attribute 'linkalways'} 
{attribute 'no_explicit_call' := 'This FB is a CLASS and must be accessed using methods or properties'}
{attribute 'enable_dynamic_creation'}
FUNCTION_BLOCK FINAL MODTURNS_LREAL EXTENDS Node
VAR
	value : _LREAL(0.0);
	arg : _LREAL(0.0);
	out : _DINT(0);
END_VAR

METHOD FB_init : BOOL
VAR_INPUT
	bInitRetains : BOOL; // if TRUE, the retain variables are initialized (warm start / cold start)
	bInCopyCode : BOOL;  // if TRUE, the instance afterwards gets moved into the copy code (online change)
END_VAR
AddInput('value',THIS^.value);
AddInput('arg',THIS^.arg);
AddOutput('out', THIS^.out);
END_METHOD

METHOD PUBLIC Clone : I_Node
VAR
	pNode : POINTER TO MODTURNS_LREAL;
END_VAR
pNode := __NEW(MODTURNS_LREAL);
Clone := pNode^;
END_METHOD

METHOD PROTECTED OnExecute
VAR
END_VAR
out.Value := MODTURNS(value.Value, arg.Value);
END_METHOD

END_FUNCTION_BLOCK

// Advanced/Nodes/SIN/SIN_LREAL
{attribute 'linkalways'} 
{attribute 'no_explicit_call' := 'This FB is a CLASS and must be accessed using methods or properties'}
{attribute 'enable_dynamic_creation'}
FUNCTION_BLOCK FINAL SIN_LREAL EXTENDS Node
VAR
	in : _LREAL(0.0);
	out : _LREAL(0.0);
END_VAR

METHOD FB_init : BOOL
VAR_INPUT
	bInitRetains : BOOL; // if TRUE, the retain variables are initialized (warm start / cold start)
	bInCopyCode : BOOL;  // if TRUE, the instance afterwards gets moved into the copy code (online change)
END_VAR
AddInput('in',THIS^.in);
AddOutput('out', THIS^.out);
END_METHOD

METHOD PUBLIC Clone : I_Node
VAR
	pNode : POINTER TO SIN_LREAL;
END_VAR
pNode := __NEW(SIN_LREAL);
Clone := pNode^;
END_METHOD

METHOD PROTECTED OnExecute
VAR
END_VAR
out.Value := SIN(in.Value);
END_METHOD

END_FUNCTION_BLOCK

// Advanced/Nodes/SQRT/SQRT_LREAL
{attribute 'linkalways'} 
{attribute 'no_explicit_call' := 'This FB is a CLASS and must be accessed using methods or properties'}
{attribute 'enable_dynamic_creation'}
FUNCTION_BLOCK FINAL SQRT_LREAL EXTENDS Node
VAR
	in : _LREAL(0.0);
	out : _LREAL(0.0);
END_VAR

METHOD FB_init : BOOL
VAR_INPUT
	bInitRetains : BOOL; // if TRUE, the retain variables are initialized (warm start / cold start)
	bInCopyCode : BOOL;  // if TRUE, the instance afterwards gets moved into the copy code (online change)
END_VAR
AddInput('in',THIS^.in);
AddOutput('out', THIS^.out);
END_METHOD

METHOD PUBLIC Clone : I_Node
VAR
	pNode : POINTER TO SQRT_LREAL;
END_VAR
pNode := __NEW(SQRT_LREAL);
Clone := pNode^;
END_METHOD

METHOD PROTECTED OnExecute
VAR
END_VAR
out.Value := SQRT(in.Value);
END_METHOD

END_FUNCTION_BLOCK

// Advanced/Nodes/TAN/TAN_LREAL
{attribute 'linkalways'} 
{attribute 'no_explicit_call' := 'This FB is a CLASS and must be accessed using methods or properties'}
{attribute 'enable_dynamic_creation'}
FUNCTION_BLOCK FINAL TAN_LREAL EXTENDS Node
VAR
	in : _LREAL(0.0);
	out : _LREAL(0.0);
END_VAR

METHOD FB_init : BOOL
VAR_INPUT
	bInitRetains : BOOL; // if TRUE, the retain variables are initialized (warm start / cold start)
	bInCopyCode : BOOL;  // if TRUE, the instance afterwards gets moved into the copy code (online change)
END_VAR
AddInput('in',THIS^.in);
AddOutput('out', THIS^.out);
END_METHOD

METHOD PUBLIC Clone : I_Node
VAR
	pNode : POINTER TO TAN_LREAL;
END_VAR
pNode := __NEW(TAN_LREAL);
Clone := pNode^;
END_METHOD

METHOD PROTECTED OnExecute
VAR
END_VAR
out.Value := TAN(in.Value);
END_METHOD

END_FUNCTION_BLOCK

// Advanced/Nodes/TRUNC/TRUNC_LREAL
{attribute 'linkalways'} 
{attribute 'no_explicit_call' := 'This FB is a CLASS and must be accessed using methods or properties'}
{attribute 'enable_dynamic_creation'}
FUNCTION_BLOCK FINAL TRUNC_LREAL EXTENDS Node
VAR
	in : _LREAL(0.0);
	out : _LREAL(0.0);
END_VAR

METHOD FB_init : BOOL
VAR_INPUT
	bInitRetains : BOOL; // if TRUE, the retain variables are initialized (warm start / cold start)
	bInCopyCode : BOOL;  // if TRUE, the instance afterwards gets moved into the copy code (online change)
END_VAR
AddInput('in',THIS^.in);
AddOutput('out', THIS^.out);
END_METHOD

METHOD PUBLIC Clone : I_Node
VAR
	pNode : POINTER TO TRUNC_LREAL;
END_VAR
pNode := __NEW(TRUNC_LREAL);
Clone := pNode^;
END_METHOD

METHOD PROTECTED OnExecute
VAR
END_VAR
out.Value := LTRUNC(in.Value);
END_METHOD

END_FUNCTION_BLOCK

// Advanced/Nodes/MathAdvancedPack
{attribute 'linkalways'} 
{attribute 'no_explicit_call' := 'This FB is a CLASS and must be accessed using methods or properties'}
{attribute 'enable_dynamic_creation'}
FUNCTION_BLOCK MathAdvancedPack IMPLEMENTS I_GraphPack
VAR
	ABS_BYTE : ABS_BYTE;
	ABS_DINT : ABS_DINT;
	ABS_DWORD : ABS_DWORD;
	ABS_INT : ABS_INT;
	ABS_LINT : ABS_LINT;
	ABS_LREAL : ABS_LREAL;
	ABS_LWORD : ABS_LWORD;
	ABS_REAL : ABS_REAL;
	ABS_SINT : ABS_SINT;
	ABS_UDINT : ABS_UDINT;
	ABS_UINT : ABS_UINT;
	ABS_ULINT : ABS_ULINT;
	ABS_USINT : ABS_USINT;
	ABS_WORD : ABS_WORD;
	
	ACOS_LREAL : ACOS_LREAL;
	ASIN_LREAL : ASIN_LREAL;
	ATAN_LREAL : ATAN_LREAL;
	COS_LREAL : COS_LREAL;
	SIN_LREAL : SIN_LREAL;
	TAN_LREAL : TAN_LREAL;
	
	EXP_LREAL : EXP_LREAL;
	EXPT_LREAL : EXPT_LREAL;
	FLOOR_LREAL : FLOOR_LREAL;
	FRAC_LREAL : FRAC_LREAL;
	LN_LREAL : LN_LREAL;
	LOG_LREAL : LOG_LREAL;
	SQRT_LREAL : SQRT_LREAL;
	TRUNC_LREAL : TRUNC_LREAL;
	MODABS_LREAL : MODABS_LREAL;
END_VAR

METHOD Register
VAR_INPUT
	Datatypes : I_Datatypes;
	NodeFactory : I_NodeFactory;
END_VAR
NodeFactory.AddNodeAsPrototype('Math/Advanced/ABS/ABS_BYTE',ABS_BYTE);
NodeFactory.AddNodeAsPrototype('Math/Advanced/ABS/ABS_DINT',ABS_DINT);
NodeFactory.AddNodeAsPrototype('Math/Advanced/ABS/ABS_DWORD',ABS_DWORD);
NodeFactory.AddNodeAsPrototype('Math/Advanced/ABS/ABS_INT',ABS_INT);
NodeFactory.AddNodeAsPrototype('Math/Advanced/ABS/ABS_LINT',ABS_LINT);
NodeFactory.AddNodeAsPrototype('Math/Advanced/ABS/ABS_LREAL',ABS_LREAL);
NodeFactory.AddNodeAsPrototype('Math/Advanced/ABS/ABS_LWORD',ABS_LWORD);
NodeFactory.AddNodeAsPrototype('Math/Advanced/ABS/ABS_REAL',ABS_REAL);
NodeFactory.AddNodeAsPrototype('Math/Advanced/ABS/ABS_SINT',ABS_SINT);
NodeFactory.AddNodeAsPrototype('Math/Advanced/ABS/ABS_UDINT',ABS_UDINT);
NodeFactory.AddNodeAsPrototype('Math/Advanced/ABS/ABS_UINT',ABS_UINT);
NodeFactory.AddNodeAsPrototype('Math/Advanced/ABS/ABS_ULINT',ABS_ULINT);
NodeFactory.AddNodeAsPrototype('Math/Advanced/ABS/ABS_USINT',ABS_USINT);
NodeFactory.AddNodeAsPrototype('Math/Advanced/ABS/ABS_WORD',ABS_WORD);

NodeFactory.AddNodeAsPrototype('Math/Advanced/ACOS/ACOS_LREAL',ACOS_LREAL);
NodeFactory.AddNodeAsPrototype('Math/Advanced/ASIN/ASIN_LREAL',ASIN_LREAL);
NodeFactory.AddNodeAsPrototype('Math/Advanced/ATAN/ATAN_LREAL',ATAN_LREAL);
NodeFactory.AddNodeAsPrototype('Math/Advanced/COS/COS_LREAL',COS_LREAL);
NodeFactory.AddNodeAsPrototype('Math/Advanced/SIN/SIN_LREAL',SIN_LREAL);
NodeFactory.AddNodeAsPrototype('Math/Advanced/TAN/TAN_LREAL',TAN_LREAL);

NodeFactory.AddNodeAsPrototype('Math/Advanced/EXP/EXP_LREAL',EXP_LREAL);
NodeFactory.AddNodeAsPrototype('Math/Advanced/EXPT/EXPT_LREAL',EXPT_LREAL);
NodeFactory.AddNodeAsPrototype('Math/Advanced/FLOOR/FLOOR_LREAL',FLOOR_LREAL);
NodeFactory.AddNodeAsPrototype('Math/Advanced/FRAC/FRAC_LREAL',FRAC_LREAL);
NodeFactory.AddNodeAsPrototype('Math/Advanced/LN/LN_LREAL',LN_LREAL);
NodeFactory.AddNodeAsPrototype('Math/Advanced/LOG/LOG_LREAL',LOG_LREAL);
NodeFactory.AddNodeAsPrototype('Math/Advanced/SQRT/SQRT_LREAL',SQRT_LREAL);
NodeFactory.AddNodeAsPrototype('Math/Advanced/TRUNC/TRUNC_LREAL',TRUNC_LREAL);
NodeFactory.AddNodeAsPrototype('Math/Advanced/MODABS/MODABS_LREAL',MODABS_LREAL);
END_METHOD

END_FUNCTION_BLOCK

// Comparison/Nodes/EQ/EQ_BYTE
{attribute 'linkalways'} 
{attribute 'no_explicit_call' := 'This FB is a CLASS and must be accessed using methods or properties'}
{attribute 'enable_dynamic_creation'}
FUNCTION_BLOCK FINAL EQ_BYTE EXTENDS Node
VAR
	in1 : _BYTE(0);
	in2 : _BYTE(0);
	out : _BOOL(FALSE);
END_VAR

METHOD FB_init : BOOL
VAR_INPUT
	bInitRetains : BOOL; // if TRUE, the retain variables are initialized (warm start / cold start)
	bInCopyCode : BOOL;  // if TRUE, the instance afterwards gets moved into the copy code (online change)
END_VAR
AddInput('in1',THIS^.in1);
AddInput('in2',THIS^.in2);
AddOutput('out', THIS^.out);
END_METHOD

METHOD PUBLIC Clone : I_Node
VAR
	pNode : POINTER TO EQ_BYTE;
END_VAR
pNode := __NEW(EQ_BYTE);
Clone := pNode^;
END_METHOD

METHOD PROTECTED OnExecute
VAR
END_VAR
out.Value := in1.Value = in2.Value;
END_METHOD

END_FUNCTION_BLOCK

// Comparison/Nodes/EQ/EQ_DINT
{attribute 'linkalways'} 
{attribute 'no_explicit_call' := 'This FB is a CLASS and must be accessed using methods or properties'}
{attribute 'enable_dynamic_creation'}
FUNCTION_BLOCK FINAL EQ_DINT EXTENDS Node
VAR
	in1 : _DINT(0);
	in2 : _DINT(0);
	out : _BOOL(FALSE);
END_VAR

METHOD FB_init : BOOL
VAR_INPUT
	bInitRetains : BOOL; // if TRUE, the retain variables are initialized (warm start / cold start)
	bInCopyCode : BOOL;  // if TRUE, the instance afterwards gets moved into the copy code (online change)
END_VAR
AddInput('in1',THIS^.in1);
AddInput('in2',THIS^.in2);
AddOutput('out', THIS^.out);
END_METHOD

METHOD PUBLIC Clone : I_Node
VAR
	pNode : POINTER TO EQ_DINT;
END_VAR
pNode := __NEW(EQ_DINT);
Clone := pNode^;
END_METHOD

METHOD PROTECTED OnExecute
VAR
END_VAR
out.Value := in1.Value = in2.Value;
END_METHOD

END_FUNCTION_BLOCK

// Comparison/Nodes/EQ/EQ_DWORD
{attribute 'linkalways'} 
{attribute 'no_explicit_call' := 'This FB is a CLASS and must be accessed using methods or properties'}
{attribute 'enable_dynamic_creation'}
FUNCTION_BLOCK FINAL EQ_DWORD EXTENDS Node
VAR
	in1 : _DWORD(0);
	in2 : _DWORD(0);
	out : _BOOL(FALSE);
END_VAR

METHOD FB_init : BOOL
VAR_INPUT
	bInitRetains : BOOL; // if TRUE, the retain variables are initialized (warm start / cold start)
	bInCopyCode : BOOL;  // if TRUE, the instance afterwards gets moved into the copy code (online change)
END_VAR
AddInput('in1',THIS^.in1);
AddInput('in2',THIS^.in2);
AddOutput('out', THIS^.out);
END_METHOD

METHOD PUBLIC Clone : I_Node
VAR
	pNode : POINTER TO EQ_DWORD;
END_VAR
pNode := __NEW(EQ_DWORD);
Clone := pNode^;
END_METHOD

METHOD PROTECTED OnExecute
VAR
END_VAR
out.Value := in1.Value = in2.Value;
END_METHOD

END_FUNCTION_BLOCK

// Comparison/Nodes/EQ/EQ_INT
{attribute 'linkalways'} 
{attribute 'no_explicit_call' := 'This FB is a CLASS and must be accessed using methods or properties'}
{attribute 'enable_dynamic_creation'}
FUNCTION_BLOCK FINAL EQ_INT EXTENDS Node
VAR
	in1 : _INT(0);
	in2 : _INT(0);
	out : _BOOL(FALSE);
END_VAR

METHOD FB_init : BOOL
VAR_INPUT
	bInitRetains : BOOL; // if TRUE, the retain variables are initialized (warm start / cold start)
	bInCopyCode : BOOL;  // if TRUE, the instance afterwards gets moved into the copy code (online change)
END_VAR
AddInput('in1',THIS^.in1);
AddInput('in2',THIS^.in2);
AddOutput('out', THIS^.out);
END_METHOD

METHOD PUBLIC Clone : I_Node
VAR
	pNode : POINTER TO EQ_INT;
END_VAR
pNode := __NEW(EQ_INT);
Clone := pNode^;
END_METHOD

METHOD PROTECTED OnExecute
VAR
END_VAR
out.Value := in1.Value = in2.Value;
END_METHOD

END_FUNCTION_BLOCK

// Comparison/Nodes/EQ/EQ_LINT
{attribute 'linkalways'} 
{attribute 'no_explicit_call' := 'This FB is a CLASS and must be accessed using methods or properties'}
{attribute 'enable_dynamic_creation'}
FUNCTION_BLOCK FINAL EQ_LINT EXTENDS Node
VAR
	in1 : _LINT(0);
	in2 : _LINT(0);
	out : _BOOL(FALSE);
END_VAR

METHOD FB_init : BOOL
VAR_INPUT
	bInitRetains : BOOL; // if TRUE, the retain variables are initialized (warm start / cold start)
	bInCopyCode : BOOL;  // if TRUE, the instance afterwards gets moved into the copy code (online change)
END_VAR
AddInput('in1',THIS^.in1);
AddInput('in2',THIS^.in2);
AddOutput('out', THIS^.out);
END_METHOD

METHOD PUBLIC Clone : I_Node
VAR
	pNode : POINTER TO EQ_LINT;
END_VAR
pNode := __NEW(EQ_LINT);
Clone := pNode^;
END_METHOD

METHOD PROTECTED OnExecute
VAR
END_VAR
out.Value := in1.Value = in2.Value;
END_METHOD

END_FUNCTION_BLOCK

// Comparison/Nodes/EQ/EQ_LREAL
{attribute 'linkalways'} 
{attribute 'no_explicit_call' := 'This FB is a CLASS and must be accessed using methods or properties'}
{attribute 'enable_dynamic_creation'}
FUNCTION_BLOCK FINAL EQ_LREAL EXTENDS Node
VAR
	in1 : _LREAL(0.0);
	in2 : _LREAL(0.0);
	out : _BOOL(FALSE);
END_VAR

METHOD FB_init : BOOL
VAR_INPUT
	bInitRetains : BOOL; // if TRUE, the retain variables are initialized (warm start / cold start)
	bInCopyCode : BOOL;  // if TRUE, the instance afterwards gets moved into the copy code (online change)
END_VAR
AddInput('in1',THIS^.in1);
AddInput('in2',THIS^.in2);
AddOutput('out', THIS^.out);
END_METHOD

METHOD PUBLIC Clone : I_Node
VAR
	pNode : POINTER TO EQ_LREAL;
END_VAR
pNode := __NEW(EQ_LREAL);
Clone := pNode^;
END_METHOD

METHOD PROTECTED OnExecute
VAR
END_VAR
out.Value := in1.Value = in2.Value;
END_METHOD

END_FUNCTION_BLOCK

// Comparison/Nodes/EQ/EQ_LWORD
{attribute 'linkalways'} 
{attribute 'no_explicit_call' := 'This FB is a CLASS and must be accessed using methods or properties'}
{attribute 'enable_dynamic_creation'}
FUNCTION_BLOCK FINAL EQ_LWORD EXTENDS Node
VAR
	in1 : _LWORD(0);
	in2 : _LWORD(0);
	out : _BOOL(FALSE);
END_VAR

METHOD FB_init : BOOL
VAR_INPUT
	bInitRetains : BOOL; // if TRUE, the retain variables are initialized (warm start / cold start)
	bInCopyCode : BOOL;  // if TRUE, the instance afterwards gets moved into the copy code (online change)
END_VAR
AddInput('in1',THIS^.in1);
AddInput('in2',THIS^.in2);
AddOutput('out', THIS^.out);
END_METHOD

METHOD PUBLIC Clone : I_Node
VAR
	pNode : POINTER TO EQ_LWORD;
END_VAR
pNode := __NEW(EQ_LWORD);
Clone := pNode^;
END_METHOD

METHOD PROTECTED OnExecute
VAR
END_VAR
out.Value := in1.Value = in2.Value;
END_METHOD

END_FUNCTION_BLOCK

// Comparison/Nodes/EQ/EQ_REAL
{attribute 'linkalways'} 
{attribute 'no_explicit_call' := 'This FB is a CLASS and must be accessed using methods or properties'}
{attribute 'enable_dynamic_creation'}
FUNCTION_BLOCK FINAL EQ_REAL EXTENDS Node
VAR
	in1 : _REAL(0.0);
	in2 : _REAL(0.0);
	out : _BOOL(FALSE);
END_VAR

METHOD FB_init : BOOL
VAR_INPUT
	bInitRetains : BOOL; // if TRUE, the retain variables are initialized (warm start / cold start)
	bInCopyCode : BOOL;  // if TRUE, the instance afterwards gets moved into the copy code (online change)
END_VAR
AddInput('in1',THIS^.in1);
AddInput('in2',THIS^.in2);
AddOutput('out', THIS^.out);
END_METHOD

METHOD PUBLIC Clone : I_Node
VAR
	pNode : POINTER TO EQ_REAL;
END_VAR
pNode := __NEW(EQ_REAL);
Clone := pNode^;
END_METHOD

METHOD PROTECTED OnExecute
VAR
END_VAR
out.Value := in1.Value = in2.Value;
END_METHOD

END_FUNCTION_BLOCK

// Comparison/Nodes/EQ/EQ_SINT
{attribute 'linkalways'} 
{attribute 'no_explicit_call' := 'This FB is a CLASS and must be accessed using methods or properties'}
{attribute 'enable_dynamic_creation'}
FUNCTION_BLOCK FINAL EQ_SINT EXTENDS Node
VAR
	in1 : _SINT(0);
	in2 : _SINT(0);
	out : _BOOL(FALSE);
END_VAR

METHOD FB_init : BOOL
VAR_INPUT
	bInitRetains : BOOL; // if TRUE, the retain variables are initialized (warm start / cold start)
	bInCopyCode : BOOL;  // if TRUE, the instance afterwards gets moved into the copy code (online change)
END_VAR
AddInput('in1',THIS^.in1);
AddInput('in2',THIS^.in2);
AddOutput('out', THIS^.out);
END_METHOD

METHOD PUBLIC Clone : I_Node
VAR
	pNode : POINTER TO EQ_SINT;
END_VAR
pNode := __NEW(EQ_SINT);
Clone := pNode^;
END_METHOD

METHOD PROTECTED OnExecute
VAR
END_VAR
out.Value := in1.Value = in2.Value;
END_METHOD

END_FUNCTION_BLOCK

// Comparison/Nodes/EQ/EQ_UDINT
{attribute 'linkalways'} 
{attribute 'no_explicit_call' := 'This FB is a CLASS and must be accessed using methods or properties'}
{attribute 'enable_dynamic_creation'}
FUNCTION_BLOCK FINAL EQ_UDINT EXTENDS Node
VAR
	in1 : _UDINT(0);
	in2 : _UDINT(0);
	out : _BOOL(FALSE);
END_VAR

METHOD FB_init : BOOL
VAR_INPUT
	bInitRetains : BOOL; // if TRUE, the retain variables are initialized (warm start / cold start)
	bInCopyCode : BOOL;  // if TRUE, the instance afterwards gets moved into the copy code (online change)
END_VAR
AddInput('in1',THIS^.in1);
AddInput('in2',THIS^.in2);
AddOutput('out', THIS^.out);
END_METHOD

METHOD PUBLIC Clone : I_Node
VAR
	pNode : POINTER TO EQ_UDINT;
END_VAR
pNode := __NEW(EQ_UDINT);
Clone := pNode^;
END_METHOD

METHOD PROTECTED OnExecute
VAR
END_VAR
out.Value := in1.Value = in2.Value;
END_METHOD

END_FUNCTION_BLOCK

// Comparison/Nodes/EQ/EQ_UINT
{attribute 'linkalways'} 
{attribute 'no_explicit_call' := 'This FB is a CLASS and must be accessed using methods or properties'}
{attribute 'enable_dynamic_creation'}
FUNCTION_BLOCK FINAL EQ_UINT EXTENDS Node
VAR
	in1 : _UINT(0);
	in2 : _UINT(0);
	out : _BOOL(FALSE);
END_VAR

METHOD FB_init : BOOL
VAR_INPUT
	bInitRetains : BOOL; // if TRUE, the retain variables are initialized (warm start / cold start)
	bInCopyCode : BOOL;  // if TRUE, the instance afterwards gets moved into the copy code (online change)
END_VAR
AddInput('in1',THIS^.in1);
AddInput('in2',THIS^.in2);
AddOutput('out', THIS^.out);
END_METHOD

METHOD PUBLIC Clone : I_Node
VAR
	pNode : POINTER TO EQ_UINT;
END_VAR
pNode := __NEW(EQ_UINT);
Clone := pNode^;
END_METHOD

METHOD PROTECTED OnExecute
VAR
END_VAR
out.Value := in1.Value = in2.Value;
END_METHOD

END_FUNCTION_BLOCK

// Comparison/Nodes/EQ/EQ_ULINT
{attribute 'linkalways'} 
{attribute 'no_explicit_call' := 'This FB is a CLASS and must be accessed using methods or properties'}
{attribute 'enable_dynamic_creation'}
FUNCTION_BLOCK FINAL EQ_ULINT EXTENDS Node
VAR
	in1 : _ULINT(0);
	in2 : _ULINT(0);
	out : _BOOL(FALSE);
END_VAR

METHOD FB_init : BOOL
VAR_INPUT
	bInitRetains : BOOL; // if TRUE, the retain variables are initialized (warm start / cold start)
	bInCopyCode : BOOL;  // if TRUE, the instance afterwards gets moved into the copy code (online change)
END_VAR
AddInput('in1',THIS^.in1);
AddInput('in2',THIS^.in2);
AddOutput('out', THIS^.out);
END_METHOD

METHOD PUBLIC Clone : I_Node
VAR
	pNode : POINTER TO EQ_ULINT;
END_VAR
pNode := __NEW(EQ_ULINT);
Clone := pNode^;
END_METHOD

METHOD PROTECTED OnExecute
VAR
END_VAR
out.Value := in1.Value = in2.Value;
END_METHOD

END_FUNCTION_BLOCK

// Comparison/Nodes/EQ/EQ_USINT
{attribute 'linkalways'} 
{attribute 'no_explicit_call' := 'This FB is a CLASS and must be accessed using methods or properties'}
{attribute 'enable_dynamic_creation'}
FUNCTION_BLOCK FINAL EQ_USINT EXTENDS Node
VAR
	in1 : _USINT(0);
	in2 : _USINT(0);
	out : _BOOL(FALSE);
END_VAR

METHOD FB_init : BOOL
VAR_INPUT
	bInitRetains : BOOL; // if TRUE, the retain variables are initialized (warm start / cold start)
	bInCopyCode : BOOL;  // if TRUE, the instance afterwards gets moved into the copy code (online change)
END_VAR
AddInput('in1',THIS^.in1);
AddInput('in2',THIS^.in2);
AddOutput('out', THIS^.out);
END_METHOD

METHOD PUBLIC Clone : I_Node
VAR
	pNode : POINTER TO EQ_USINT;
END_VAR
pNode := __NEW(EQ_USINT);
Clone := pNode^;
END_METHOD

METHOD PROTECTED OnExecute
VAR
END_VAR
out.Value := in1.Value = in2.Value;
END_METHOD

END_FUNCTION_BLOCK

// Comparison/Nodes/EQ/EQ_WORD
{attribute 'linkalways'} 
{attribute 'no_explicit_call' := 'This FB is a CLASS and must be accessed using methods or properties'}
{attribute 'enable_dynamic_creation'}
FUNCTION_BLOCK FINAL EQ_WORD EXTENDS Node
VAR
	in1 : _WORD(0);
	in2 : _WORD(0);
	out : _BOOL(FALSE);
END_VAR

METHOD FB_init : BOOL
VAR_INPUT
	bInitRetains : BOOL; // if TRUE, the retain variables are initialized (warm start / cold start)
	bInCopyCode : BOOL;  // if TRUE, the instance afterwards gets moved into the copy code (online change)
END_VAR
AddInput('in1',THIS^.in1);
AddInput('in2',THIS^.in2);
AddOutput('out', THIS^.out);
END_METHOD

METHOD PUBLIC Clone : I_Node
VAR
	pNode : POINTER TO EQ_WORD;
END_VAR
pNode := __NEW(EQ_WORD);
Clone := pNode^;
END_METHOD

METHOD PROTECTED OnExecute
VAR
END_VAR
out.Value := in1.Value = in2.Value;
END_METHOD

END_FUNCTION_BLOCK

// Comparison/Nodes/GE/GE_BYTE
{attribute 'linkalways'} 
{attribute 'no_explicit_call' := 'This FB is a CLASS and must be accessed using methods or properties'}
{attribute 'enable_dynamic_creation'}
FUNCTION_BLOCK FINAL GE_BYTE EXTENDS Node
VAR
	in1 : _BYTE(0);
	in2 : _BYTE(0);
	out : _BOOL(FALSE);
END_VAR

METHOD FB_init : BOOL
VAR_INPUT
	bInitRetains : BOOL; // if TRUE, the retain variables are initialized (warm start / cold start)
	bInCopyCode : BOOL;  // if TRUE, the instance afterwards gets moved into the copy code (online change)
END_VAR
AddInput('in1',THIS^.in1);
AddInput('in2',THIS^.in2);
AddOutput('out', THIS^.out);
END_METHOD

METHOD PUBLIC Clone : I_Node
VAR
	pNode : POINTER TO GE_BYTE;
END_VAR
pNode := __NEW(GE_BYTE);
Clone := pNode^;
END_METHOD

METHOD PROTECTED OnExecute
VAR
END_VAR
out.Value := in1.Value >= in2.Value;
END_METHOD

END_FUNCTION_BLOCK

// Comparison/Nodes/GE/GE_DINT
{attribute 'linkalways'} 
{attribute 'no_explicit_call' := 'This FB is a CLASS and must be accessed using methods or properties'}
{attribute 'enable_dynamic_creation'}
FUNCTION_BLOCK FINAL GE_DINT EXTENDS Node
VAR
	in1 : _DINT(0);
	in2 : _DINT(0);
	out : _BOOL(FALSE);
END_VAR

METHOD FB_init : BOOL
VAR_INPUT
	bInitRetains : BOOL; // if TRUE, the retain variables are initialized (warm start / cold start)
	bInCopyCode : BOOL;  // if TRUE, the instance afterwards gets moved into the copy code (online change)
END_VAR
AddInput('in1',THIS^.in1);
AddInput('in2',THIS^.in2);
AddOutput('out', THIS^.out);
END_METHOD

METHOD PUBLIC Clone : I_Node
VAR
	pNode : POINTER TO GE_DINT;
END_VAR
pNode := __NEW(GE_DINT);
Clone := pNode^;
END_METHOD

METHOD PROTECTED OnExecute
VAR
END_VAR
out.Value := in1.Value >= in2.Value;
END_METHOD

END_FUNCTION_BLOCK

// Comparison/Nodes/GE/GE_DWORD
{attribute 'linkalways'} 
{attribute 'no_explicit_call' := 'This FB is a CLASS and must be accessed using methods or properties'}
{attribute 'enable_dynamic_creation'}
FUNCTION_BLOCK FINAL GE_DWORD EXTENDS Node
VAR
	in1 : _DWORD(0);
	in2 : _DWORD(0);
	out : _BOOL(FALSE);
END_VAR

METHOD FB_init : BOOL
VAR_INPUT
	bInitRetains : BOOL; // if TRUE, the retain variables are initialized (warm start / cold start)
	bInCopyCode : BOOL;  // if TRUE, the instance afterwards gets moved into the copy code (online change)
END_VAR
AddInput('in1',THIS^.in1);
AddInput('in2',THIS^.in2);
AddOutput('out', THIS^.out);
END_METHOD

METHOD PUBLIC Clone : I_Node
VAR
	pNode : POINTER TO GE_DWORD;
END_VAR
pNode := __NEW(GE_DWORD);
Clone := pNode^;
END_METHOD

METHOD PROTECTED OnExecute
VAR
END_VAR
out.Value := in1.Value >= in2.Value;
END_METHOD

END_FUNCTION_BLOCK

// Comparison/Nodes/GE/GE_INT
{attribute 'linkalways'} 
{attribute 'no_explicit_call' := 'This FB is a CLASS and must be accessed using methods or properties'}
{attribute 'enable_dynamic_creation'}
FUNCTION_BLOCK FINAL GE_INT EXTENDS Node
VAR
	in1 : _INT(0);
	in2 : _INT(0);
	out : _BOOL(FALSE);
END_VAR

METHOD FB_init : BOOL
VAR_INPUT
	bInitRetains : BOOL; // if TRUE, the retain variables are initialized (warm start / cold start)
	bInCopyCode : BOOL;  // if TRUE, the instance afterwards gets moved into the copy code (online change)
END_VAR
AddInput('in1',THIS^.in1);
AddInput('in2',THIS^.in2);
AddOutput('out', THIS^.out);
END_METHOD

METHOD PUBLIC Clone : I_Node
VAR
	pNode : POINTER TO GE_INT;
END_VAR
pNode := __NEW(GE_INT);
Clone := pNode^;
END_METHOD

METHOD PROTECTED OnExecute
VAR
END_VAR
out.Value := in1.Value >= in2.Value;
END_METHOD

END_FUNCTION_BLOCK

// Comparison/Nodes/GE/GE_LINT
{attribute 'linkalways'} 
{attribute 'no_explicit_call' := 'This FB is a CLASS and must be accessed using methods or properties'}
{attribute 'enable_dynamic_creation'}
FUNCTION_BLOCK FINAL GE_LINT EXTENDS Node
VAR
	in1 : _LINT(0);
	in2 : _LINT(0);
	out : _BOOL(FALSE);
END_VAR

METHOD FB_init : BOOL
VAR_INPUT
	bInitRetains : BOOL; // if TRUE, the retain variables are initialized (warm start / cold start)
	bInCopyCode : BOOL;  // if TRUE, the instance afterwards gets moved into the copy code (online change)
END_VAR
AddInput('in1',THIS^.in1);
AddInput('in2',THIS^.in2);
AddOutput('out', THIS^.out);
END_METHOD

METHOD PUBLIC Clone : I_Node
VAR
	pNode : POINTER TO GE_LINT;
END_VAR
pNode := __NEW(GE_LINT);
Clone := pNode^;
END_METHOD

METHOD PROTECTED OnExecute
VAR
END_VAR
out.Value := in1.Value >= in2.Value;
END_METHOD

END_FUNCTION_BLOCK

// Comparison/Nodes/GE/GE_LREAL
{attribute 'linkalways'} 
{attribute 'no_explicit_call' := 'This FB is a CLASS and must be accessed using methods or properties'}
{attribute 'enable_dynamic_creation'}
FUNCTION_BLOCK FINAL GE_LREAL EXTENDS Node
VAR
	in1 : _LREAL(0.0);
	in2 : _LREAL(0.0);
	out : _BOOL(FALSE);
END_VAR

METHOD FB_init : BOOL
VAR_INPUT
	bInitRetains : BOOL; // if TRUE, the retain variables are initialized (warm start / cold start)
	bInCopyCode : BOOL;  // if TRUE, the instance afterwards gets moved into the copy code (online change)
END_VAR
AddInput('in1',THIS^.in1);
AddInput('in2',THIS^.in2);
AddOutput('out', THIS^.out);
END_METHOD

METHOD PUBLIC Clone : I_Node
VAR
	pNode : POINTER TO GE_LREAL;
END_VAR
pNode := __NEW(GE_LREAL);
Clone := pNode^;
END_METHOD

METHOD PROTECTED OnExecute
VAR
END_VAR
out.Value := in1.Value >= in2.Value;
END_METHOD

END_FUNCTION_BLOCK

// Comparison/Nodes/GE/GE_LWORD
{attribute 'linkalways'} 
{attribute 'no_explicit_call' := 'This FB is a CLASS and must be accessed using methods or properties'}
{attribute 'enable_dynamic_creation'}
FUNCTION_BLOCK FINAL GE_LWORD EXTENDS Node
VAR
	in1 : _LWORD(0);
	in2 : _LWORD(0);
	out : _BOOL(FALSE);
END_VAR

METHOD FB_init : BOOL
VAR_INPUT
	bInitRetains : BOOL; // if TRUE, the retain variables are initialized (warm start / cold start)
	bInCopyCode : BOOL;  // if TRUE, the instance afterwards gets moved into the copy code (online change)
END_VAR
AddInput('in1',THIS^.in1);
AddInput('in2',THIS^.in2);
AddOutput('out', THIS^.out);
END_METHOD

METHOD PUBLIC Clone : I_Node
VAR
	pNode : POINTER TO GE_LWORD;
END_VAR
pNode := __NEW(GE_LWORD);
Clone := pNode^;
END_METHOD

METHOD PROTECTED OnExecute
VAR
END_VAR
out.Value := in1.Value >= in2.Value;
END_METHOD

END_FUNCTION_BLOCK

// Comparison/Nodes/GE/GE_REAL
{attribute 'linkalways'} 
{attribute 'no_explicit_call' := 'This FB is a CLASS and must be accessed using methods or properties'}
{attribute 'enable_dynamic_creation'}
FUNCTION_BLOCK FINAL GE_REAL EXTENDS Node
VAR
	in1 : _REAL(0.0);
	in2 : _REAL(0.0);
	out : _BOOL(FALSE);
END_VAR

METHOD FB_init : BOOL
VAR_INPUT
	bInitRetains : BOOL; // if TRUE, the retain variables are initialized (warm start / cold start)
	bInCopyCode : BOOL;  // if TRUE, the instance afterwards gets moved into the copy code (online change)
END_VAR
AddInput('in1',THIS^.in1);
AddInput('in2',THIS^.in2);
AddOutput('out', THIS^.out);
END_METHOD

METHOD PUBLIC Clone : I_Node
VAR
	pNode : POINTER TO GE_REAL;
END_VAR
pNode := __NEW(GE_REAL);
Clone := pNode^;
END_METHOD

METHOD PROTECTED OnExecute
VAR
END_VAR
out.Value := in1.Value >= in2.Value;
END_METHOD

END_FUNCTION_BLOCK

// Comparison/Nodes/GE/GE_SINT
{attribute 'linkalways'} 
{attribute 'no_explicit_call' := 'This FB is a CLASS and must be accessed using methods or properties'}
{attribute 'enable_dynamic_creation'}
FUNCTION_BLOCK FINAL GE_SINT EXTENDS Node
VAR
	in1 : _SINT(0);
	in2 : _SINT(0);
	out : _BOOL(FALSE);
END_VAR

METHOD FB_init : BOOL
VAR_INPUT
	bInitRetains : BOOL; // if TRUE, the retain variables are initialized (warm start / cold start)
	bInCopyCode : BOOL;  // if TRUE, the instance afterwards gets moved into the copy code (online change)
END_VAR
AddInput('in1',THIS^.in1);
AddInput('in2',THIS^.in2);
AddOutput('out', THIS^.out);
END_METHOD

METHOD PUBLIC Clone : I_Node
VAR
	pNode : POINTER TO GE_SINT;
END_VAR
pNode := __NEW(GE_SINT);
Clone := pNode^;
END_METHOD

METHOD PROTECTED OnExecute
VAR
END_VAR
out.Value := in1.Value >= in2.Value;
END_METHOD

END_FUNCTION_BLOCK

// Comparison/Nodes/GE/GE_UDINT
{attribute 'linkalways'} 
{attribute 'no_explicit_call' := 'This FB is a CLASS and must be accessed using methods or properties'}
{attribute 'enable_dynamic_creation'}
FUNCTION_BLOCK FINAL GE_UDINT EXTENDS Node
VAR
	in1 : _UDINT(0);
	in2 : _UDINT(0);
	out : _BOOL(FALSE);
END_VAR

METHOD FB_init : BOOL
VAR_INPUT
	bInitRetains : BOOL; // if TRUE, the retain variables are initialized (warm start / cold start)
	bInCopyCode : BOOL;  // if TRUE, the instance afterwards gets moved into the copy code (online change)
END_VAR
AddInput('in1',THIS^.in1);
AddInput('in2',THIS^.in2);
AddOutput('out', THIS^.out);
END_METHOD

METHOD PUBLIC Clone : I_Node
VAR
	pNode : POINTER TO GE_UDINT;
END_VAR
pNode := __NEW(GE_UDINT);
Clone := pNode^;
END_METHOD

METHOD PROTECTED OnExecute
VAR
END_VAR
out.Value := in1.Value >= in2.Value;
END_METHOD

END_FUNCTION_BLOCK

// Comparison/Nodes/GE/GE_UINT
{attribute 'linkalways'} 
{attribute 'no_explicit_call' := 'This FB is a CLASS and must be accessed using methods or properties'}
{attribute 'enable_dynamic_creation'}
FUNCTION_BLOCK FINAL GE_UINT EXTENDS Node
VAR
	in1 : _UINT(0);
	in2 : _UINT(0);
	out : _BOOL(FALSE);
END_VAR

METHOD FB_init : BOOL
VAR_INPUT
	bInitRetains : BOOL; // if TRUE, the retain variables are initialized (warm start / cold start)
	bInCopyCode : BOOL;  // if TRUE, the instance afterwards gets moved into the copy code (online change)
END_VAR
AddInput('in1',THIS^.in1);
AddInput('in2',THIS^.in2);
AddOutput('out', THIS^.out);
END_METHOD

METHOD PUBLIC Clone : I_Node
VAR
	pNode : POINTER TO GE_UINT;
END_VAR
pNode := __NEW(GE_UINT);
Clone := pNode^;
END_METHOD

METHOD PROTECTED OnExecute
VAR
END_VAR
out.Value := in1.Value >= in2.Value;
END_METHOD

END_FUNCTION_BLOCK

// Comparison/Nodes/GE/GE_ULINT
{attribute 'linkalways'} 
{attribute 'no_explicit_call' := 'This FB is a CLASS and must be accessed using methods or properties'}
{attribute 'enable_dynamic_creation'}
FUNCTION_BLOCK FINAL GE_ULINT EXTENDS Node
VAR
	in1 : _ULINT(0);
	in2 : _ULINT(0);
	out : _BOOL(FALSE);
END_VAR

METHOD FB_init : BOOL
VAR_INPUT
	bInitRetains : BOOL; // if TRUE, the retain variables are initialized (warm start / cold start)
	bInCopyCode : BOOL;  // if TRUE, the instance afterwards gets moved into the copy code (online change)
END_VAR
AddInput('in1',THIS^.in1);
AddInput('in2',THIS^.in2);
AddOutput('out', THIS^.out);
END_METHOD

METHOD PUBLIC Clone : I_Node
VAR
	pNode : POINTER TO GE_ULINT;
END_VAR
pNode := __NEW(GE_ULINT);
Clone := pNode^;
END_METHOD

METHOD PROTECTED OnExecute
VAR
END_VAR
out.Value := in1.Value >= in2.Value;
END_METHOD

END_FUNCTION_BLOCK

// Comparison/Nodes/GE/GE_USINT
{attribute 'linkalways'} 
{attribute 'no_explicit_call' := 'This FB is a CLASS and must be accessed using methods or properties'}
{attribute 'enable_dynamic_creation'}
FUNCTION_BLOCK FINAL GE_USINT EXTENDS Node
VAR
	in1 : _USINT(0);
	in2 : _USINT(0);
	out : _BOOL(FALSE);
END_VAR

METHOD FB_init : BOOL
VAR_INPUT
	bInitRetains : BOOL; // if TRUE, the retain variables are initialized (warm start / cold start)
	bInCopyCode : BOOL;  // if TRUE, the instance afterwards gets moved into the copy code (online change)
END_VAR
AddInput('in1',THIS^.in1);
AddInput('in2',THIS^.in2);
AddOutput('out', THIS^.out);
END_METHOD

METHOD PUBLIC Clone : I_Node
VAR
	pNode : POINTER TO GE_USINT;
END_VAR
pNode := __NEW(GE_USINT);
Clone := pNode^;
END_METHOD

METHOD PROTECTED OnExecute
VAR
END_VAR
out.Value := in1.Value >= in2.Value;
END_METHOD

END_FUNCTION_BLOCK

// Comparison/Nodes/GE/GE_WORD
{attribute 'linkalways'} 
{attribute 'no_explicit_call' := 'This FB is a CLASS and must be accessed using methods or properties'}
{attribute 'enable_dynamic_creation'}
FUNCTION_BLOCK FINAL GE_WORD EXTENDS Node
VAR
	in1 : _WORD(0);
	in2 : _WORD(0);
	out : _BOOL(FALSE);
END_VAR

METHOD FB_init : BOOL
VAR_INPUT
	bInitRetains : BOOL; // if TRUE, the retain variables are initialized (warm start / cold start)
	bInCopyCode : BOOL;  // if TRUE, the instance afterwards gets moved into the copy code (online change)
END_VAR
AddInput('in1',THIS^.in1);
AddInput('in2',THIS^.in2);
AddOutput('out', THIS^.out);
END_METHOD

METHOD PUBLIC Clone : I_Node
VAR
	pNode : POINTER TO GE_WORD;
END_VAR
pNode := __NEW(GE_WORD);
Clone := pNode^;
END_METHOD

METHOD PROTECTED OnExecute
VAR
END_VAR
out.Value := in1.Value >= in2.Value;
END_METHOD

END_FUNCTION_BLOCK

// Comparison/Nodes/GT/GT_BYTE
{attribute 'linkalways'} 
{attribute 'no_explicit_call' := 'This FB is a CLASS and must be accessed using methods or properties'}
{attribute 'enable_dynamic_creation'}
FUNCTION_BLOCK FINAL GT_BYTE EXTENDS Node
VAR
	in1 : _BYTE(0);
	in2 : _BYTE(0);
	out : _BOOL(FALSE);
END_VAR

METHOD FB_init : BOOL
VAR_INPUT
	bInitRetains : BOOL; // if TRUE, the retain variables are initialized (warm start / cold start)
	bInCopyCode : BOOL;  // if TRUE, the instance afterwards gets moved into the copy code (online change)
END_VAR
AddInput('in1',THIS^.in1);
AddInput('in2',THIS^.in2);
AddOutput('out', THIS^.out);
END_METHOD

METHOD PUBLIC Clone : I_Node
VAR
	pNode : POINTER TO GT_BYTE;
END_VAR
pNode := __NEW(GT_BYTE);
Clone := pNode^;
END_METHOD

METHOD PROTECTED OnExecute
VAR
END_VAR
out.Value := in1.Value > in2.Value;
END_METHOD

END_FUNCTION_BLOCK

// Comparison/Nodes/GT/GT_DINT
{attribute 'linkalways'} 
{attribute 'no_explicit_call' := 'This FB is a CLASS and must be accessed using methods or properties'}
{attribute 'enable_dynamic_creation'}
FUNCTION_BLOCK FINAL GT_DINT EXTENDS Node
VAR
	in1 : _DINT(0);
	in2 : _DINT(0);
	out : _BOOL(FALSE);
END_VAR

METHOD FB_init : BOOL
VAR_INPUT
	bInitRetains : BOOL; // if TRUE, the retain variables are initialized (warm start / cold start)
	bInCopyCode : BOOL;  // if TRUE, the instance afterwards gets moved into the copy code (online change)
END_VAR
AddInput('in1',THIS^.in1);
AddInput('in2',THIS^.in2);
AddOutput('out', THIS^.out);
END_METHOD

METHOD PUBLIC Clone : I_Node
VAR
	pNode : POINTER TO GT_DINT;
END_VAR
pNode := __NEW(GT_DINT);
Clone := pNode^;
END_METHOD

METHOD PROTECTED OnExecute
VAR
END_VAR
out.Value := in1.Value > in2.Value;
END_METHOD

END_FUNCTION_BLOCK

// Comparison/Nodes/GT/GT_DWORD
{attribute 'linkalways'} 
{attribute 'no_explicit_call' := 'This FB is a CLASS and must be accessed using methods or properties'}
{attribute 'enable_dynamic_creation'}
FUNCTION_BLOCK FINAL GT_DWORD EXTENDS Node
VAR
	in1 : _DWORD(0);
	in2 : _DWORD(0);
	out : _BOOL(FALSE);
END_VAR

METHOD FB_init : BOOL
VAR_INPUT
	bInitRetains : BOOL; // if TRUE, the retain variables are initialized (warm start / cold start)
	bInCopyCode : BOOL;  // if TRUE, the instance afterwards gets moved into the copy code (online change)
END_VAR
AddInput('in1',THIS^.in1);
AddInput('in2',THIS^.in2);
AddOutput('out', THIS^.out);
END_METHOD

METHOD PUBLIC Clone : I_Node
VAR
	pNode : POINTER TO GT_DWORD;
END_VAR
pNode := __NEW(GT_DWORD);
Clone := pNode^;
END_METHOD

METHOD PROTECTED OnExecute
VAR
END_VAR
out.Value := in1.Value > in2.Value;
END_METHOD

END_FUNCTION_BLOCK

// Comparison/Nodes/GT/GT_INT
{attribute 'linkalways'} 
{attribute 'no_explicit_call' := 'This FB is a CLASS and must be accessed using methods or properties'}
{attribute 'enable_dynamic_creation'}
FUNCTION_BLOCK FINAL GT_INT EXTENDS Node
VAR
	in1 : _INT(0);
	in2 : _INT(0);
	out : _BOOL(FALSE);
END_VAR

METHOD FB_init : BOOL
VAR_INPUT
	bInitRetains : BOOL; // if TRUE, the retain variables are initialized (warm start / cold start)
	bInCopyCode : BOOL;  // if TRUE, the instance afterwards gets moved into the copy code (online change)
END_VAR
AddInput('in1',THIS^.in1);
AddInput('in2',THIS^.in2);
AddOutput('out', THIS^.out);
END_METHOD

METHOD PUBLIC Clone : I_Node
VAR
	pNode : POINTER TO GT_INT;
END_VAR
pNode := __NEW(GT_INT);
Clone := pNode^;
END_METHOD

METHOD PROTECTED OnExecute
VAR
END_VAR
out.Value := in1.Value > in2.Value;
END_METHOD

END_FUNCTION_BLOCK

// Comparison/Nodes/GT/GT_LINT
{attribute 'linkalways'} 
{attribute 'no_explicit_call' := 'This FB is a CLASS and must be accessed using methods or properties'}
{attribute 'enable_dynamic_creation'}
FUNCTION_BLOCK FINAL GT_LINT EXTENDS Node
VAR
	in1 : _LINT(0);
	in2 : _LINT(0);
	out : _BOOL(FALSE);
END_VAR

METHOD FB_init : BOOL
VAR_INPUT
	bInitRetains : BOOL; // if TRUE, the retain variables are initialized (warm start / cold start)
	bInCopyCode : BOOL;  // if TRUE, the instance afterwards gets moved into the copy code (online change)
END_VAR
AddInput('in1',THIS^.in1);
AddInput('in2',THIS^.in2);
AddOutput('out', THIS^.out);
END_METHOD

METHOD PUBLIC Clone : I_Node
VAR
	pNode : POINTER TO GT_LINT;
END_VAR
pNode := __NEW(GT_LINT);
Clone := pNode^;
END_METHOD

METHOD PROTECTED OnExecute
VAR
END_VAR
out.Value := in1.Value > in2.Value;
END_METHOD

END_FUNCTION_BLOCK

// Comparison/Nodes/GT/GT_LREAL
{attribute 'linkalways'} 
{attribute 'no_explicit_call' := 'This FB is a CLASS and must be accessed using methods or properties'}
{attribute 'enable_dynamic_creation'}
FUNCTION_BLOCK FINAL GT_LREAL EXTENDS Node
VAR
	in1 : _LREAL(0.0);
	in2 : _LREAL(0.0);
	out : _BOOL(FALSE);
END_VAR

METHOD FB_init : BOOL
VAR_INPUT
	bInitRetains : BOOL; // if TRUE, the retain variables are initialized (warm start / cold start)
	bInCopyCode : BOOL;  // if TRUE, the instance afterwards gets moved into the copy code (online change)
END_VAR
AddInput('in1',THIS^.in1);
AddInput('in2',THIS^.in2);
AddOutput('out', THIS^.out);
END_METHOD

METHOD PUBLIC Clone : I_Node
VAR
	pNode : POINTER TO GT_LREAL;
END_VAR
pNode := __NEW(GT_LREAL);
Clone := pNode^;
END_METHOD

METHOD PROTECTED OnExecute
VAR
END_VAR
out.Value := in1.Value > in2.Value;
END_METHOD

END_FUNCTION_BLOCK

// Comparison/Nodes/GT/GT_LWORD
{attribute 'linkalways'} 
{attribute 'no_explicit_call' := 'This FB is a CLASS and must be accessed using methods or properties'}
{attribute 'enable_dynamic_creation'}
FUNCTION_BLOCK FINAL GT_LWORD EXTENDS Node
VAR
	in1 : _LWORD(0);
	in2 : _LWORD(0);
	out : _BOOL(FALSE);
END_VAR

METHOD FB_init : BOOL
VAR_INPUT
	bInitRetains : BOOL; // if TRUE, the retain variables are initialized (warm start / cold start)
	bInCopyCode : BOOL;  // if TRUE, the instance afterwards gets moved into the copy code (online change)
END_VAR
AddInput('in1',THIS^.in1);
AddInput('in2',THIS^.in2);
AddOutput('out', THIS^.out);
END_METHOD

METHOD PUBLIC Clone : I_Node
VAR
	pNode : POINTER TO GT_LWORD;
END_VAR
pNode := __NEW(GT_LWORD);
Clone := pNode^;
END_METHOD

METHOD PROTECTED OnExecute
VAR
END_VAR
out.Value := in1.Value > in2.Value;
END_METHOD

END_FUNCTION_BLOCK

// Comparison/Nodes/GT/GT_REAL
{attribute 'linkalways'} 
{attribute 'no_explicit_call' := 'This FB is a CLASS and must be accessed using methods or properties'}
{attribute 'enable_dynamic_creation'}
FUNCTION_BLOCK FINAL GT_REAL EXTENDS Node
VAR
	in1 : _REAL(0.0);
	in2 : _REAL(0.0);
	out : _BOOL(FALSE);
END_VAR

METHOD FB_init : BOOL
VAR_INPUT
	bInitRetains : BOOL; // if TRUE, the retain variables are initialized (warm start / cold start)
	bInCopyCode : BOOL;  // if TRUE, the instance afterwards gets moved into the copy code (online change)
END_VAR
AddInput('in1',THIS^.in1);
AddInput('in2',THIS^.in2);
AddOutput('out', THIS^.out);
END_METHOD

METHOD PUBLIC Clone : I_Node
VAR
	pNode : POINTER TO GT_REAL;
END_VAR
pNode := __NEW(GT_REAL);
Clone := pNode^;
END_METHOD

METHOD PROTECTED OnExecute
VAR
END_VAR
out.Value := in1.Value > in2.Value;
END_METHOD

END_FUNCTION_BLOCK

// Comparison/Nodes/GT/GT_SINT
{attribute 'linkalways'} 
{attribute 'no_explicit_call' := 'This FB is a CLASS and must be accessed using methods or properties'}
{attribute 'enable_dynamic_creation'}
FUNCTION_BLOCK FINAL GT_SINT EXTENDS Node
VAR
	in1 : _SINT(0);
	in2 : _SINT(0);
	out : _BOOL(FALSE);
END_VAR

METHOD FB_init : BOOL
VAR_INPUT
	bInitRetains : BOOL; // if TRUE, the retain variables are initialized (warm start / cold start)
	bInCopyCode : BOOL;  // if TRUE, the instance afterwards gets moved into the copy code (online change)
END_VAR
AddInput('in1',THIS^.in1);
AddInput('in2',THIS^.in2);
AddOutput('out', THIS^.out);
END_METHOD

METHOD PUBLIC Clone : I_Node
VAR
	pNode : POINTER TO GT_SINT;
END_VAR
pNode := __NEW(GT_SINT);
Clone := pNode^;
END_METHOD

METHOD PROTECTED OnExecute
VAR
END_VAR
out.Value := in1.Value > in2.Value;
END_METHOD

END_FUNCTION_BLOCK

// Comparison/Nodes/GT/GT_UDINT
{attribute 'linkalways'} 
{attribute 'no_explicit_call' := 'This FB is a CLASS and must be accessed using methods or properties'}
{attribute 'enable_dynamic_creation'}
FUNCTION_BLOCK FINAL GT_UDINT EXTENDS Node
VAR
	in1 : _UDINT(0);
	in2 : _UDINT(0);
	out : _BOOL(FALSE);
END_VAR

METHOD FB_init : BOOL
VAR_INPUT
	bInitRetains : BOOL; // if TRUE, the retain variables are initialized (warm start / cold start)
	bInCopyCode : BOOL;  // if TRUE, the instance afterwards gets moved into the copy code (online change)
END_VAR
AddInput('in1',THIS^.in1);
AddInput('in2',THIS^.in2);
AddOutput('out', THIS^.out);
END_METHOD

METHOD PUBLIC Clone : I_Node
VAR
	pNode : POINTER TO GT_UDINT;
END_VAR
pNode := __NEW(GT_UDINT);
Clone := pNode^;
END_METHOD

METHOD PROTECTED OnExecute
VAR
END_VAR
out.Value := in1.Value > in2.Value;
END_METHOD

END_FUNCTION_BLOCK

// Comparison/Nodes/GT/GT_UINT
{attribute 'linkalways'} 
{attribute 'no_explicit_call' := 'This FB is a CLASS and must be accessed using methods or properties'}
{attribute 'enable_dynamic_creation'}
FUNCTION_BLOCK FINAL GT_UINT EXTENDS Node
VAR
	in1 : _UINT(0);
	in2 : _UINT(0);
	out : _BOOL(FALSE);
END_VAR

METHOD FB_init : BOOL
VAR_INPUT
	bInitRetains : BOOL; // if TRUE, the retain variables are initialized (warm start / cold start)
	bInCopyCode : BOOL;  // if TRUE, the instance afterwards gets moved into the copy code (online change)
END_VAR
AddInput('in1',THIS^.in1);
AddInput('in2',THIS^.in2);
AddOutput('out', THIS^.out);
END_METHOD

METHOD PUBLIC Clone : I_Node
VAR
	pNode : POINTER TO GT_UINT;
END_VAR
pNode := __NEW(GT_UINT);
Clone := pNode^;
END_METHOD

METHOD PROTECTED OnExecute
VAR
END_VAR
out.Value := in1.Value > in2.Value;
END_METHOD

END_FUNCTION_BLOCK

// Comparison/Nodes/GT/GT_ULINT
{attribute 'linkalways'} 
{attribute 'no_explicit_call' := 'This FB is a CLASS and must be accessed using methods or properties'}
{attribute 'enable_dynamic_creation'}
FUNCTION_BLOCK FINAL GT_ULINT EXTENDS Node
VAR
	in1 : _ULINT(0);
	in2 : _ULINT(0);
	out : _BOOL(FALSE);
END_VAR

METHOD FB_init : BOOL
VAR_INPUT
	bInitRetains : BOOL; // if TRUE, the retain variables are initialized (warm start / cold start)
	bInCopyCode : BOOL;  // if TRUE, the instance afterwards gets moved into the copy code (online change)
END_VAR
AddInput('in1',THIS^.in1);
AddInput('in2',THIS^.in2);
AddOutput('out', THIS^.out);
END_METHOD

METHOD PUBLIC Clone : I_Node
VAR
	pNode : POINTER TO GT_ULINT;
END_VAR
pNode := __NEW(GT_ULINT);
Clone := pNode^;
END_METHOD

METHOD PROTECTED OnExecute
VAR
END_VAR
out.Value := in1.Value > in2.Value;
END_METHOD

END_FUNCTION_BLOCK

// Comparison/Nodes/GT/GT_USINT
{attribute 'linkalways'} 
{attribute 'no_explicit_call' := 'This FB is a CLASS and must be accessed using methods or properties'}
{attribute 'enable_dynamic_creation'}
FUNCTION_BLOCK FINAL GT_USINT EXTENDS Node
VAR
	in1 : _USINT(0);
	in2 : _USINT(0);
	out : _BOOL(FALSE);
END_VAR

METHOD FB_init : BOOL
VAR_INPUT
	bInitRetains : BOOL; // if TRUE, the retain variables are initialized (warm start / cold start)
	bInCopyCode : BOOL;  // if TRUE, the instance afterwards gets moved into the copy code (online change)
END_VAR
AddInput('in1',THIS^.in1);
AddInput('in2',THIS^.in2);
AddOutput('out', THIS^.out);
END_METHOD

METHOD PUBLIC Clone : I_Node
VAR
	pNode : POINTER TO GT_USINT;
END_VAR
pNode := __NEW(GT_USINT);
Clone := pNode^;
END_METHOD

METHOD PROTECTED OnExecute
VAR
END_VAR
out.Value := in1.Value > in2.Value;
END_METHOD

END_FUNCTION_BLOCK

// Comparison/Nodes/GT/GT_WORD
{attribute 'linkalways'} 
{attribute 'no_explicit_call' := 'This FB is a CLASS and must be accessed using methods or properties'}
{attribute 'enable_dynamic_creation'}
FUNCTION_BLOCK FINAL GT_WORD EXTENDS Node
VAR
	in1 : _WORD(0);
	in2 : _WORD(0);
	out : _BOOL(FALSE);
END_VAR

METHOD FB_init : BOOL
VAR_INPUT
	bInitRetains : BOOL; // if TRUE, the retain variables are initialized (warm start / cold start)
	bInCopyCode : BOOL;  // if TRUE, the instance afterwards gets moved into the copy code (online change)
END_VAR
AddInput('in1',THIS^.in1);
AddInput('in2',THIS^.in2);
AddOutput('out', THIS^.out);
END_METHOD

METHOD PUBLIC Clone : I_Node
VAR
	pNode : POINTER TO GT_WORD;
END_VAR
pNode := __NEW(GT_WORD);
Clone := pNode^;
END_METHOD

METHOD PROTECTED OnExecute
VAR
END_VAR
out.Value := in1.Value > in2.Value;
END_METHOD

END_FUNCTION_BLOCK

// Comparison/Nodes/LE/LE_BYTE
{attribute 'linkalways'} 
{attribute 'no_explicit_call' := 'This FB is a CLASS and must be accessed using methods or properties'}
{attribute 'enable_dynamic_creation'}
FUNCTION_BLOCK FINAL LE_BYTE EXTENDS Node
VAR
	in1 : _BYTE(0);
	in2 : _BYTE(0);
	out : _BOOL(FALSE);
END_VAR

METHOD FB_init : BOOL
VAR_INPUT
	bInitRetains : BOOL; // if TRUE, the retain variables are initialized (warm start / cold start)
	bInCopyCode : BOOL;  // if TRUE, the instance afterwards gets moved into the copy code (online change)
END_VAR
AddInput('in1',THIS^.in1);
AddInput('in2',THIS^.in2);
AddOutput('out', THIS^.out);
END_METHOD

METHOD PUBLIC Clone : I_Node
VAR
	pNode : POINTER TO LE_BYTE;
END_VAR
pNode := __NEW(LE_BYTE);
Clone := pNode^;
END_METHOD

METHOD PROTECTED OnExecute
VAR
END_VAR
out.Value := in1.Value <= in2.Value;
END_METHOD

END_FUNCTION_BLOCK

// Comparison/Nodes/LE/LE_DINT
{attribute 'linkalways'} 
{attribute 'no_explicit_call' := 'This FB is a CLASS and must be accessed using methods or properties'}
{attribute 'enable_dynamic_creation'}
FUNCTION_BLOCK FINAL LE_DINT EXTENDS Node
VAR
	in1 : _DINT(0);
	in2 : _DINT(0);
	out : _BOOL(FALSE);
END_VAR

METHOD FB_init : BOOL
VAR_INPUT
	bInitRetains : BOOL; // if TRUE, the retain variables are initialized (warm start / cold start)
	bInCopyCode : BOOL;  // if TRUE, the instance afterwards gets moved into the copy code (online change)
END_VAR
AddInput('in1',THIS^.in1);
AddInput('in2',THIS^.in2);
AddOutput('out', THIS^.out);
END_METHOD

METHOD PUBLIC Clone : I_Node
VAR
	pNode : POINTER TO LE_DINT;
END_VAR
pNode := __NEW(LE_DINT);
Clone := pNode^;
END_METHOD

METHOD PROTECTED OnExecute
VAR
END_VAR
out.Value := in1.Value <= in2.Value;
END_METHOD

END_FUNCTION_BLOCK

// Comparison/Nodes/LE/LE_DWORD
{attribute 'linkalways'} 
{attribute 'no_explicit_call' := 'This FB is a CLASS and must be accessed using methods or properties'}
{attribute 'enable_dynamic_creation'}
FUNCTION_BLOCK FINAL LE_DWORD EXTENDS Node
VAR
	in1 : _DWORD(0);
	in2 : _DWORD(0);
	out : _BOOL(FALSE);
END_VAR

METHOD FB_init : BOOL
VAR_INPUT
	bInitRetains : BOOL; // if TRUE, the retain variables are initialized (warm start / cold start)
	bInCopyCode : BOOL;  // if TRUE, the instance afterwards gets moved into the copy code (online change)
END_VAR
AddInput('in1',THIS^.in1);
AddInput('in2',THIS^.in2);
AddOutput('out', THIS^.out);
END_METHOD

METHOD PUBLIC Clone : I_Node
VAR
	pNode : POINTER TO LE_DWORD;
END_VAR
pNode := __NEW(LE_DWORD);
Clone := pNode^;
END_METHOD

METHOD PROTECTED OnExecute
VAR
END_VAR
out.Value := in1.Value <= in2.Value;
END_METHOD

END_FUNCTION_BLOCK

// Comparison/Nodes/LE/LE_INT
{attribute 'linkalways'} 
{attribute 'no_explicit_call' := 'This FB is a CLASS and must be accessed using methods or properties'}
{attribute 'enable_dynamic_creation'}
FUNCTION_BLOCK FINAL LE_INT EXTENDS Node
VAR
	in1 : _INT(0);
	in2 : _INT(0);
	out : _BOOL(FALSE);
END_VAR

METHOD FB_init : BOOL
VAR_INPUT
	bInitRetains : BOOL; // if TRUE, the retain variables are initialized (warm start / cold start)
	bInCopyCode : BOOL;  // if TRUE, the instance afterwards gets moved into the copy code (online change)
END_VAR
AddInput('in1',THIS^.in1);
AddInput('in2',THIS^.in2);
AddOutput('out', THIS^.out);
END_METHOD

METHOD PUBLIC Clone : I_Node
VAR
	pNode : POINTER TO LE_INT;
END_VAR
pNode := __NEW(LE_INT);
Clone := pNode^;
END_METHOD

METHOD PROTECTED OnExecute
VAR
END_VAR
out.Value := in1.Value <= in2.Value;
END_METHOD

END_FUNCTION_BLOCK

// Comparison/Nodes/LE/LE_LINT
{attribute 'linkalways'} 
{attribute 'no_explicit_call' := 'This FB is a CLASS and must be accessed using methods or properties'}
{attribute 'enable_dynamic_creation'}
FUNCTION_BLOCK FINAL LE_LINT EXTENDS Node
VAR
	in1 : _LINT(0);
	in2 : _LINT(0);
	out : _BOOL(FALSE);
END_VAR

METHOD FB_init : BOOL
VAR_INPUT
	bInitRetains : BOOL; // if TRUE, the retain variables are initialized (warm start / cold start)
	bInCopyCode : BOOL;  // if TRUE, the instance afterwards gets moved into the copy code (online change)
END_VAR
AddInput('in1',THIS^.in1);
AddInput('in2',THIS^.in2);
AddOutput('out', THIS^.out);
END_METHOD

METHOD PUBLIC Clone : I_Node
VAR
	pNode : POINTER TO LE_LINT;
END_VAR
pNode := __NEW(LE_LINT);
Clone := pNode^;
END_METHOD

METHOD PROTECTED OnExecute
VAR
END_VAR
out.Value := in1.Value <= in2.Value;
END_METHOD

END_FUNCTION_BLOCK

// Comparison/Nodes/LE/LE_LREAL
{attribute 'linkalways'} 
{attribute 'no_explicit_call' := 'This FB is a CLASS and must be accessed using methods or properties'}
{attribute 'enable_dynamic_creation'}
FUNCTION_BLOCK FINAL LE_LREAL EXTENDS Node
VAR
	in1 : _LREAL(0.0);
	in2 : _LREAL(0.0);
	out : _BOOL(FALSE);
END_VAR

METHOD FB_init : BOOL
VAR_INPUT
	bInitRetains : BOOL; // if TRUE, the retain variables are initialized (warm start / cold start)
	bInCopyCode : BOOL;  // if TRUE, the instance afterwards gets moved into the copy code (online change)
END_VAR
AddInput('in1',THIS^.in1);
AddInput('in2',THIS^.in2);
AddOutput('out', THIS^.out);
END_METHOD

METHOD PUBLIC Clone : I_Node
VAR
	pNode : POINTER TO LE_LREAL;
END_VAR
pNode := __NEW(LE_LREAL);
Clone := pNode^;
END_METHOD

METHOD PROTECTED OnExecute
VAR
END_VAR
out.Value := in1.Value <= in2.Value;
END_METHOD

END_FUNCTION_BLOCK

// Comparison/Nodes/LE/LE_LWORD
{attribute 'linkalways'} 
{attribute 'no_explicit_call' := 'This FB is a CLASS and must be accessed using methods or properties'}
{attribute 'enable_dynamic_creation'}
FUNCTION_BLOCK FINAL LE_LWORD EXTENDS Node
VAR
	in1 : _LWORD(0);
	in2 : _LWORD(0);
	out : _BOOL(FALSE);
END_VAR

METHOD FB_init : BOOL
VAR_INPUT
	bInitRetains : BOOL; // if TRUE, the retain variables are initialized (warm start / cold start)
	bInCopyCode : BOOL;  // if TRUE, the instance afterwards gets moved into the copy code (online change)
END_VAR
AddInput('in1',THIS^.in1);
AddInput('in2',THIS^.in2);
AddOutput('out', THIS^.out);
END_METHOD

METHOD PUBLIC Clone : I_Node
VAR
	pNode : POINTER TO LE_LWORD;
END_VAR
pNode := __NEW(LE_LWORD);
Clone := pNode^;
END_METHOD

METHOD PROTECTED OnExecute
VAR
END_VAR
out.Value := in1.Value <= in2.Value;
END_METHOD

END_FUNCTION_BLOCK

// Comparison/Nodes/LE/LE_REAL
{attribute 'linkalways'} 
{attribute 'no_explicit_call' := 'This FB is a CLASS and must be accessed using methods or properties'}
{attribute 'enable_dynamic_creation'}
FUNCTION_BLOCK FINAL LE_REAL EXTENDS Node
VAR
	in1 : _REAL(0.0);
	in2 : _REAL(0.0);
	out : _BOOL(FALSE);
END_VAR

METHOD FB_init : BOOL
VAR_INPUT
	bInitRetains : BOOL; // if TRUE, the retain variables are initialized (warm start / cold start)
	bInCopyCode : BOOL;  // if TRUE, the instance afterwards gets moved into the copy code (online change)
END_VAR
AddInput('in1',THIS^.in1);
AddInput('in2',THIS^.in2);
AddOutput('out', THIS^.out);
END_METHOD

METHOD PUBLIC Clone : I_Node
VAR
	pNode : POINTER TO LE_REAL;
END_VAR
pNode := __NEW(LE_REAL);
Clone := pNode^;
END_METHOD

METHOD PROTECTED OnExecute
VAR
END_VAR
out.Value := in1.Value <= in2.Value;
END_METHOD

END_FUNCTION_BLOCK

// Comparison/Nodes/LE/LE_SINT
{attribute 'linkalways'} 
{attribute 'no_explicit_call' := 'This FB is a CLASS and must be accessed using methods or properties'}
{attribute 'enable_dynamic_creation'}
FUNCTION_BLOCK FINAL LE_SINT EXTENDS Node
VAR
	in1 : _SINT(0);
	in2 : _SINT(0);
	out : _BOOL(FALSE);
END_VAR

METHOD FB_init : BOOL
VAR_INPUT
	bInitRetains : BOOL; // if TRUE, the retain variables are initialized (warm start / cold start)
	bInCopyCode : BOOL;  // if TRUE, the instance afterwards gets moved into the copy code (online change)
END_VAR
AddInput('in1',THIS^.in1);
AddInput('in2',THIS^.in2);
AddOutput('out', THIS^.out);
END_METHOD

METHOD PUBLIC Clone : I_Node
VAR
	pNode : POINTER TO LE_SINT;
END_VAR
pNode := __NEW(LE_SINT);
Clone := pNode^;
END_METHOD

METHOD PROTECTED OnExecute
VAR
END_VAR
out.Value := in1.Value <= in2.Value;
END_METHOD

END_FUNCTION_BLOCK

// Comparison/Nodes/LE/LE_UDINT
{attribute 'linkalways'} 
{attribute 'no_explicit_call' := 'This FB is a CLASS and must be accessed using methods or properties'}
{attribute 'enable_dynamic_creation'}
FUNCTION_BLOCK FINAL LE_UDINT EXTENDS Node
VAR
	in1 : _UDINT(0);
	in2 : _UDINT(0);
	out : _BOOL(FALSE);
END_VAR

METHOD FB_init : BOOL
VAR_INPUT
	bInitRetains : BOOL; // if TRUE, the retain variables are initialized (warm start / cold start)
	bInCopyCode : BOOL;  // if TRUE, the instance afterwards gets moved into the copy code (online change)
END_VAR
AddInput('in1',THIS^.in1);
AddInput('in2',THIS^.in2);
AddOutput('out', THIS^.out);
END_METHOD

METHOD PUBLIC Clone : I_Node
VAR
	pNode : POINTER TO LE_UDINT;
END_VAR
pNode := __NEW(LE_UDINT);
Clone := pNode^;
END_METHOD

METHOD PROTECTED OnExecute
VAR
END_VAR
out.Value := in1.Value <= in2.Value;
END_METHOD

END_FUNCTION_BLOCK

// Comparison/Nodes/LE/LE_UINT
{attribute 'linkalways'} 
{attribute 'no_explicit_call' := 'This FB is a CLASS and must be accessed using methods or properties'}
{attribute 'enable_dynamic_creation'}
FUNCTION_BLOCK FINAL LE_UINT EXTENDS Node
VAR
	in1 : _UINT(0);
	in2 : _UINT(0);
	out : _BOOL(FALSE);
END_VAR

METHOD FB_init : BOOL
VAR_INPUT
	bInitRetains : BOOL; // if TRUE, the retain variables are initialized (warm start / cold start)
	bInCopyCode : BOOL;  // if TRUE, the instance afterwards gets moved into the copy code (online change)
END_VAR
AddInput('in1',THIS^.in1);
AddInput('in2',THIS^.in2);
AddOutput('out', THIS^.out);
END_METHOD

METHOD PUBLIC Clone : I_Node
VAR
	pNode : POINTER TO LE_UINT;
END_VAR
pNode := __NEW(LE_UINT);
Clone := pNode^;
END_METHOD

METHOD PROTECTED OnExecute
VAR
END_VAR
out.Value := in1.Value <= in2.Value;
END_METHOD

END_FUNCTION_BLOCK

// Comparison/Nodes/LE/LE_ULINT
{attribute 'linkalways'} 
{attribute 'no_explicit_call' := 'This FB is a CLASS and must be accessed using methods or properties'}
{attribute 'enable_dynamic_creation'}
FUNCTION_BLOCK FINAL LE_ULINT EXTENDS Node
VAR
	in1 : _ULINT(0);
	in2 : _ULINT(0);
	out : _BOOL(FALSE);
END_VAR

METHOD FB_init : BOOL
VAR_INPUT
	bInitRetains : BOOL; // if TRUE, the retain variables are initialized (warm start / cold start)
	bInCopyCode : BOOL;  // if TRUE, the instance afterwards gets moved into the copy code (online change)
END_VAR
AddInput('in1',THIS^.in1);
AddInput('in2',THIS^.in2);
AddOutput('out', THIS^.out);
END_METHOD

METHOD PUBLIC Clone : I_Node
VAR
	pNode : POINTER TO LE_ULINT;
END_VAR
pNode := __NEW(LE_ULINT);
Clone := pNode^;
END_METHOD

METHOD PROTECTED OnExecute
VAR
END_VAR
out.Value := in1.Value <= in2.Value;
END_METHOD

END_FUNCTION_BLOCK

// Comparison/Nodes/LE/LE_USINT
{attribute 'linkalways'} 
{attribute 'no_explicit_call' := 'This FB is a CLASS and must be accessed using methods or properties'}
{attribute 'enable_dynamic_creation'}
FUNCTION_BLOCK FINAL LE_USINT EXTENDS Node
VAR
	in1 : _USINT(0);
	in2 : _USINT(0);
	out : _BOOL(FALSE);
END_VAR

METHOD FB_init : BOOL
VAR_INPUT
	bInitRetains : BOOL; // if TRUE, the retain variables are initialized (warm start / cold start)
	bInCopyCode : BOOL;  // if TRUE, the instance afterwards gets moved into the copy code (online change)
END_VAR
AddInput('in1',THIS^.in1);
AddInput('in2',THIS^.in2);
AddOutput('out', THIS^.out);
END_METHOD

METHOD PUBLIC Clone : I_Node
VAR
	pNode : POINTER TO LE_USINT;
END_VAR
pNode := __NEW(LE_USINT);
Clone := pNode^;
END_METHOD

METHOD PROTECTED OnExecute
VAR
END_VAR
out.Value := in1.Value <= in2.Value;
END_METHOD

END_FUNCTION_BLOCK

// Comparison/Nodes/LE/LE_WORD
{attribute 'linkalways'} 
{attribute 'no_explicit_call' := 'This FB is a CLASS and must be accessed using methods or properties'}
{attribute 'enable_dynamic_creation'}
FUNCTION_BLOCK FINAL LE_WORD EXTENDS Node
VAR
	in1 : _WORD(0);
	in2 : _WORD(0);
	out : _BOOL(FALSE);
END_VAR

METHOD FB_init : BOOL
VAR_INPUT
	bInitRetains : BOOL; // if TRUE, the retain variables are initialized (warm start / cold start)
	bInCopyCode : BOOL;  // if TRUE, the instance afterwards gets moved into the copy code (online change)
END_VAR
AddInput('in1',THIS^.in1);
AddInput('in2',THIS^.in2);
AddOutput('out', THIS^.out);
END_METHOD

METHOD PUBLIC Clone : I_Node
VAR
	pNode : POINTER TO LE_WORD;
END_VAR
pNode := __NEW(LE_WORD);
Clone := pNode^;
END_METHOD

METHOD PROTECTED OnExecute
VAR
END_VAR
out.Value := in1.Value <= in2.Value;
END_METHOD

END_FUNCTION_BLOCK

// Comparison/Nodes/LT/LT_BYTE
{attribute 'linkalways'} 
{attribute 'no_explicit_call' := 'This FB is a CLASS and must be accessed using methods or properties'}
{attribute 'enable_dynamic_creation'}
FUNCTION_BLOCK FINAL LT_BYTE EXTENDS Node
VAR
	in1 : _BYTE(0);
	in2 : _BYTE(0);
	out : _BOOL(FALSE);
END_VAR

METHOD FB_init : BOOL
VAR_INPUT
	bInitRetains : BOOL; // if TRUE, the retain variables are initialized (warm start / cold start)
	bInCopyCode : BOOL;  // if TRUE, the instance afterwards gets moved into the copy code (online change)
END_VAR
AddInput('in1',THIS^.in1);
AddInput('in2',THIS^.in2);
AddOutput('out', THIS^.out);
END_METHOD

METHOD PUBLIC Clone : I_Node
VAR
	pNode : POINTER TO LT_BYTE;
END_VAR
pNode := __NEW(LT_BYTE);
Clone := pNode^;
END_METHOD

METHOD PROTECTED OnExecute
VAR
END_VAR
out.Value := in1.Value < in2.Value;
END_METHOD

END_FUNCTION_BLOCK

// Comparison/Nodes/LT/LT_DINT
{attribute 'linkalways'} 
{attribute 'no_explicit_call' := 'This FB is a CLASS and must be accessed using methods or properties'}
{attribute 'enable_dynamic_creation'}
FUNCTION_BLOCK FINAL LT_DINT EXTENDS Node
VAR
	in1 : _DINT(0);
	in2 : _DINT(0);
	out : _BOOL(FALSE);
END_VAR

METHOD FB_init : BOOL
VAR_INPUT
	bInitRetains : BOOL; // if TRUE, the retain variables are initialized (warm start / cold start)
	bInCopyCode : BOOL;  // if TRUE, the instance afterwards gets moved into the copy code (online change)
END_VAR
AddInput('in1',THIS^.in1);
AddInput('in2',THIS^.in2);
AddOutput('out', THIS^.out);
END_METHOD

METHOD PUBLIC Clone : I_Node
VAR
	pNode : POINTER TO LT_DINT;
END_VAR
pNode := __NEW(LT_DINT);
Clone := pNode^;
END_METHOD

METHOD PROTECTED OnExecute
VAR
END_VAR
out.Value := in1.Value < in2.Value;
END_METHOD

END_FUNCTION_BLOCK

// Comparison/Nodes/LT/LT_DWORD
{attribute 'linkalways'} 
{attribute 'no_explicit_call' := 'This FB is a CLASS and must be accessed using methods or properties'}
{attribute 'enable_dynamic_creation'}
FUNCTION_BLOCK FINAL LT_DWORD EXTENDS Node
VAR
	in1 : _DWORD(0);
	in2 : _DWORD(0);
	out : _BOOL(FALSE);
END_VAR

METHOD FB_init : BOOL
VAR_INPUT
	bInitRetains : BOOL; // if TRUE, the retain variables are initialized (warm start / cold start)
	bInCopyCode : BOOL;  // if TRUE, the instance afterwards gets moved into the copy code (online change)
END_VAR
AddInput('in1',THIS^.in1);
AddInput('in2',THIS^.in2);
AddOutput('out', THIS^.out);
END_METHOD

METHOD PUBLIC Clone : I_Node
VAR
	pNode : POINTER TO LT_DWORD;
END_VAR
pNode := __NEW(LT_DWORD);
Clone := pNode^;
END_METHOD

METHOD PROTECTED OnExecute
VAR
END_VAR
out.Value := in1.Value < in2.Value;
END_METHOD

END_FUNCTION_BLOCK

// Comparison/Nodes/LT/LT_INT
{attribute 'linkalways'} 
{attribute 'no_explicit_call' := 'This FB is a CLASS and must be accessed using methods or properties'}
{attribute 'enable_dynamic_creation'}
FUNCTION_BLOCK FINAL LT_INT EXTENDS Node
VAR
	in1 : _INT(0);
	in2 : _INT(0);
	out : _BOOL(FALSE);
END_VAR

METHOD FB_init : BOOL
VAR_INPUT
	bInitRetains : BOOL; // if TRUE, the retain variables are initialized (warm start / cold start)
	bInCopyCode : BOOL;  // if TRUE, the instance afterwards gets moved into the copy code (online change)
END_VAR
AddInput('in1',THIS^.in1);
AddInput('in2',THIS^.in2);
AddOutput('out', THIS^.out);
END_METHOD

